LIN {X 0,Y 400.14,Z 423.786,A -85,B 0,C 180,E1 -11270.146,E2 -11270.146} C_VEL
LIN {X 0,Y 399.174,Z 418.317,A -85,B 0,C 180,E1 -11270.323,E2 -11270.323} C_VEL
LIN {X 0,Y 400.535,Z 402.133,A -85,B 0,C 180,E1 -11273.803,E2 -11273.803} C_VEL
LIN {X 0,Y 400.601,Z 399.085,A -85,B 0,C 180,E1 -11274.478,E2 -11274.478} C_VEL
LIN {X 0,Y 398.361,Z 387.399,A -85,B 0,C 180,E1 -11277.304,E2 -11277.304} C_VEL
LIN {X 0,Y 397.149,Z 382.018,A -85,B 0,C 180,E1 -11278.687,E2 -11278.687} C_VEL
LIN {X 0,Y 397.084,Z 382.025,A -85,B 0,C 180,E1 -11282.072,E2 -11282.072} C_VEL
LIN {X 0,Y 397.125,Z 382.02,A -85,B 0,C 180,E1 -11285.504,E2 -11285.504} C_VEL
LIN {X 0,Y 397.136,Z 382.02,A -85,B 0,C 180,E1 -11288.862,E2 -11288.862} C_VEL
LIN {X 0,Y 397.074,Z 382.025,A -85,B 0,C 180,E1 -11292.268,E2 -11292.268} C_VEL
LIN {X 0,Y 397.092,Z 382.023,A -85,B 0,C 180,E1 -11295.069,E2 -11295.069} C_VEL
LIN {X 0,Y 397.071,Z 382.022,A -85,B 0,C 180,E1 -11298.022,E2 -11298.022} C_VEL
LIN {X 0,Y 397.134,Z 382.018,A -85,B 0,C 180,E1 -11301.139,E2 -11301.139} C_VEL
LIN {X 0,Y 397.125,Z 382.018,A -85,B 0,C 180,E1 -11304.497,E2 -11304.497} C_VEL
LIN {X 0,Y 397.084,Z 382.02,A -85,B 0,C 180,E1 -11307.929,E2 -11307.929} C_VEL
LIN {X 0,Y 397.128,Z 382.015,A -85,B 0,C 180,E1 -11311.457,E2 -11311.457} C_VEL
LIN {X 0,Y 397.158,Z 382.011,A -85,B 0,C 180,E1 -11314.488,E2 -11314.488} C_VEL
LIN {X 0,Y 397.115,Z 382.014,A -85,B 0,C 180,E1 -11318.183,E2 -11318.183} C_VEL
LIN {X 0,Y 397.168,Z 382.003,A -85,B 0,C 180,E1 -11321.427,E2 -11321.427} C_VEL
LIN {X 0,Y 397.185,Z 382.005,A -85,B 0,C 180,E1 -11324.608,E2 -11324.608} C_VEL
LIN {X 0,Y 397.225,Z 382.004,A -85,B 0,C 180,E1 -11327.742,E2 -11327.742} C_VEL
LIN {X 0,Y 397.401,Z 381.985,A -85,B 0,C 180,E1 -11332.041,E2 -11332.041} C_VEL
LIN {X 0,Y 397.26,Z 381.999,A -85,B 0,C 180,E1 -11334.925,E2 -11334.925} C_VEL
LIN {X 0,Y 397.455,Z 381.973,A -85,B 0,C 180,E1 -11337.973,E2 -11337.973} C_VEL
LIN {X 0,Y 397.585,Z 381.959,A -85,B 0,C 180,E1 -11340,E2 -11340} C_VEL
LIN {X 0,Y 397.382,Z 381.983,A -85,B 0,C 180,E1 -11343.041,E2 -11343.041} C_VEL
LIN {X 0,Y 397.37,Z 381.983,A -85,B 0,C 180,E1 -11347.112,E2 -11347.112} C_VEL
LIN {X 0,Y 397.224,Z 382.008,A -85,B 0,C 180,E1 -11350.191,E2 -11350.191} C_VEL
LIN {X 0,Y 397.233,Z 382.005,A -85,B 0,C 180,E1 -11353.321,E2 -11353.321} C_VEL
LIN {X 0,Y 397.188,Z 382.01,A -85,B 0,C 180,E1 -11357.155,E2 -11357.155} C_VEL
LIN {X 0,Y 397.109,Z 382.019,A -85,B 0,C 180,E1 -11360.73,E2 -11360.73} C_VEL
LIN {X 0,Y 397.139,Z 382.015,A -85,B 0,C 180,E1 -11364.018,E2 -11364.018} C_VEL
LIN {X 0,Y 397.231,Z 382.12,A -85,B 0,C 180,E1 -11367.209,E2 -11367.209} C_VEL
LIN {X 0,Y 399.17,Z 392.144,A -85,B 0,C 180,E1 -11370.004,E2 -11370.004} C_VEL
LIN {X 0,Y 399.737,Z 396.779,A -85,B 0,C 180,E1 -11371.242,E2 -11371.242} C_VEL
LIN {X 0,Y 399.607,Z 398.872,A -85,B 0,C 180,E1 -11371.771,E2 -11371.771} C_VEL
LIN {X 0,Y 404.077,Z 419.363,A -85,B 0,C 180,E1 -11372.445,E2 -11372.445} C_VEL
LIN {X 0,Y 404.272,Z 424.24,A -85,B 0,C 180,E1 -11372.552,E2 -11372.552} C_VEL
LIN {X 0,Y 402.86,Z 505.983,A -85,B 0,C 180,E1 -11374.111,E2 -11374.111} C_VEL
LIN {X 0,Y 402.397,Z 518.755,A -85,B 0,C 180,E1 -11374.545,E2 -11374.545} C_VEL
LIN {X 0,Y 401.764,Z 531.63,A -85,B 0,C 180,E1 -11375.191,E2 -11375.191} C_VEL
LIN {X 0,Y 400.956,Z 543.977,A -85,B 0,C 180,E1 -11376.043,E2 -11376.043} C_VEL
LIN {X 0,Y 400.163,Z 554.558,A -85,B 0,C 180,E1 -11376.98,E2 -11376.98} C_VEL
LIN {X 0,Y 399.29,Z 565.476,A -85,B 0,C 180,E1 -11378.188,E2 -11378.188} C_VEL
LIN {X 0,Y 398.415,Z 574.461,A -85,B 0,C 180,E1 -11379.423,E2 -11379.423} C_VEL
LIN {X 0,Y 397.649,Z 582.829,A -85,B 0,C 180,E1 -11380.839,E2 -11380.839} C_VEL
LIN {X 0,Y 397.067,Z 589.697,A -85,B 0,C 180,E1 -11382.268,E2 -11382.268} C_VEL
LIN {X 0,Y 396.606,Z 595.356,A -85,B 0,C 180,E1 -11383.717,E2 -11383.717} C_VEL
LIN {X 0,Y 396.229,Z 599.96,A -85,B 0,C 180,E1 -11385.194,E2 -11385.194} C_VEL
LIN {X 0,Y 395.96,Z 603.578,A -85,B 0,C 180,E1 -11386.696,E2 -11386.696} C_VEL
LIN {X 0,Y 395.753,Z 606.265,A -85,B 0,C 180,E1 -11388.233,E2 -11388.233} C_VEL
LIN {X 0,Y 395.599,Z 608.354,A -85,B 0,C 180,E1 -11390.24,E2 -11390.24} C_VEL
LIN {X 0,Y 395.556,Z 608.831,A -85,B 0,C 180,E1 -11391.547,E2 -11391.547} C_VEL
LIN {X 0,Y 395.557,Z 608.577,A -85,B 0,C 180,E1 -11393.086,E2 -11393.086} C_VEL
LIN {X 0,Y 395.648,Z 607.213,A -85,B 0,C 180,E1 -11394.797,E2 -11394.797} C_VEL
LIN {X 0,Y 395.849,Z 604.514,A -85,B 0,C 180,E1 -11396.606,E2 -11396.606} C_VEL
LIN {X 0,Y 396.124,Z 600.493,A -85,B 0,C 180,E1 -11398.388,E2 -11398.388} C_VEL
LIN {X 0,Y 396.495,Z 594.51,A -85,B 0,C 180,E1 -11400.29,E2 -11400.29} C_VEL
LIN {X 0,Y 397.001,Z 588.053,A -85,B 0,C 180,E1 -11401.873,E2 -11401.873} C_VEL
LIN {X 0,Y 397.556,Z 581.327,A -85,B 0,C 180,E1 -11403.204,E2 -11403.204} C_VEL
LIN {X 0,Y 398.312,Z 571.9,A -85,B 0,C 180,E1 -11404.714,E2 -11404.714} C_VEL
LIN {X 0,Y 399.125,Z 562.154,A -85,B 0,C 180,E1 -11405.97,E2 -11405.97} C_VEL
LIN {X 0,Y 399.932,Z 551.066,A -85,B 0,C 180,E1 -11407.119,E2 -11407.119} C_VEL
LIN {X 0,Y 400.708,Z 539.338,A -85,B 0,C 180,E1 -11408.069,E2 -11408.069} C_VEL
LIN {X 0,Y 401.313,Z 527.263,A -85,B 0,C 180,E1 -11408.825,E2 -11408.825} C_VEL
LIN {X 0,Y 401.878,Z 514.644,A -85,B 0,C 180,E1 -11409.393,E2 -11409.393} C_VEL
LIN {X 0,Y 402.234,Z 500.536,A -85,B 0,C 180,E1 -11409.794,E2 -11409.794} C_VEL
LIN {X 0,Y 403.386,Z 420.013,A -85,B 0,C 180,E1 -11411.293,E2 -11411.293} C_VEL
LIN {X 0,Y 399.172,Z 398.042,A -85,B 0,C 180,E1 -11411.944,E2 -11411.944} C_VEL
LIN {X 0,Y 399.24,Z 393.33,A -85,B 0,C 180,E1 -11413.114,E2 -11413.114} C_VEL
LIN {X 0,Y 397.325,Z 382.653,A -85,B 0,C 180,E1 -11415.923,E2 -11415.923} C_VEL
LIN {X 0,Y 397.222,Z 382.008,A -85,B 0,C 180,E1 -11416.152,E2 -11416.152} C_VEL
LIN {X 0,Y 396.586,Z 382.088,A -85,B 0,C 180,E1 -11416.997,E2 -11416.997} C_VEL
LIN {X 0,Y 393.705,Z 382.445,A -85,B 0,C 180,E1 -11418.371,E2 -11418.371} C_VEL
LIN {X 0,Y 391.27,Z 382.745,A -85,B 0,C 180,E1 -11419.482,E2 -11419.482} C_VEL
LIN {X 0,Y 390.265,Z 382.873,A -85,B 0,C 180,E1 -11420.341,E2 -11420.341} C_VEL
LIN {X 0,Y 390.206,Z 382.88,A -85,B 0,C 180,E1 -11420.632,E2 -11420.632} C_VEL
LIN {X 0,Y 390.304,Z 382.864,A -85,B 0,C 180,E1 -11423.796,E2 -11423.796} C_VEL
LIN {X 0,Y 390.423,Z 382.851,A -85,B 0,C 180,E1 -11427.935,E2 -11427.935} C_VEL
LIN {X 0,Y 390.552,Z 382.835,A -85,B 0,C 180,E1 -11429.999,E2 -11429.999} C_VEL
LIN {X 0,Y 390.318,Z 382.862,A -85,B 0,C 180,E1 -11433.095,E2 -11433.095} C_VEL
LIN {X 0,Y 390.333,Z 382.866,A -85,B 0,C 180,E1 -11436.2,E2 -11436.2} C_VEL
LIN {X 0,Y 390.317,Z 382.867,A -85,B 0,C 180,E1 -11438.281,E2 -11438.281} C_VEL
LIN {X 0,Y 390.172,Z 382.882,A -85,B 0,C 180,E1 -11442.482,E2 -11442.482} C_VEL
LIN {X 0,Y 390.145,Z 382.886,A -85,B 0,C 180,E1 -11445.675,E2 -11445.675} C_VEL
LIN {X 0,Y 390.106,Z 382.888,A -85,B 0,C 180,E1 -11448.92,E2 -11448.92} C_VEL
LIN {X 0,Y 390.036,Z 382.9,A -85,B 0,C 180,E1 -11452.233,E2 -11452.233} C_VEL
LIN {X 0,Y 390.117,Z 382.892,A -85,B 0,C 180,E1 -11455.742,E2 -11455.742} C_VEL
LIN {X 0,Y 390.07,Z 382.893,A -85,B 0,C 180,E1 -11459.107,E2 -11459.107} C_VEL
LIN {X 0,Y 390.052,Z 382.895,A -85,B 0,C 180,E1 -11462.719,E2 -11462.719} C_VEL
LIN {X 0,Y 390.053,Z 382.899,A -85,B 0,C 180,E1 -11465.824,E2 -11465.824} C_VEL
LIN {X 0,Y 390.07,Z 382.895,A -85,B 0,C 180,E1 -11469.218,E2 -11469.218} C_VEL
LIN {X 0,Y 390.076,Z 382.892,A -85,B 0,C 180,E1 -11472.379,E2 -11472.379} C_VEL
LIN {X 0,Y 390.134,Z 383.038,A -85,B 0,C 180,E1 -11475.045,E2 -11475.045} C_VEL
LIN {X 0,Y 391.764,Z 391.926,A -85,B 0,C 180,E1 -11477.023,E2 -11477.023} C_VEL
LIN {X 0,Y 391.869,Z 396.801,A -85,B 0,C 180,E1 -11478.061,E2 -11478.061} C_VEL
LIN {X 0,Y 396.111,Z 421.486,A -85,B 0,C 180,E1 -11478.798,E2 -11478.798} C_VEL
LIN {X 0,Y 394.513,Z 506.118,A -85,B 0,C 180,E1 -11480.565,E2 -11480.565} C_VEL
LIN {X 0,Y 394.042,Z 519.35,A -85,B 0,C 180,E1 -11481.045,E2 -11481.045} C_VEL
LIN {X 0,Y 393.451,Z 532.156,A -85,B 0,C 180,E1 -11481.727,E2 -11481.727} C_VEL
LIN {X 0,Y 392.826,Z 543.595,A -85,B 0,C 180,E1 -11482.534,E2 -11482.534} C_VEL
LIN {X 0,Y 392.073,Z 555.083,A -85,B 0,C 180,E1 -11483.574,E2 -11483.574} C_VEL
LIN {X 0,Y 391.358,Z 565.608,A -85,B 0,C 180,E1 -11484.767,E2 -11484.767} C_VEL
LIN {X 0,Y 390.619,Z 575.13,A -85,B 0,C 180,E1 -11486.099,E2 -11486.099} C_VEL
LIN {X 0,Y 390.034,Z 583.947,A -85,B 0,C 180,E1 -11487.635,E2 -11487.635} C_VEL
LIN {X 0,Y 389.517,Z 590.564,A -85,B 0,C 180,E1 -11489.054,E2 -11489.054} C_VEL
LIN {X 0,Y 389.113,Z 597.059,A -85,B 0,C 180,E1 -11490.813,E2 -11490.813} C_VEL
LIN {X 0,Y 388.883,Z 601.347,A -85,B 0,C 180,E1 -11492.314,E2 -11492.314} C_VEL
LIN {X 0,Y 388.659,Z 605.419,A -85,B 0,C 180,E1 -11494.279,E2 -11494.279} C_VEL
LIN {X 0,Y 388.558,Z 607.024,A -85,B 0,C 180,E1 -11495.417,E2 -11495.417} C_VEL
LIN {X 0,Y 388.467,Z 608.568,A -85,B 0,C 180,E1 -11497.315,E2 -11497.315} C_VEL
LIN {X 0,Y 388.461,Z 608.799,A -85,B 0,C 180,E1 -11498.787,E2 -11498.787} C_VEL
LIN {X 0,Y 388.561,Z 608.285,A -85,B 0,C 180,E1 -11500.137,E2 -11500.137} C_VEL
LIN {X 0,Y 388.72,Z 606.239,A -85,B 0,C 180,E1 -11502.1,E2 -11502.1} C_VEL
LIN {X 0,Y 388.952,Z 603.258,A -85,B 0,C 180,E1 -11503.785,E2 -11503.785} C_VEL
LIN {X 0,Y 389.24,Z 599.364,A -85,B 0,C 180,E1 -11505.358,E2 -11505.358} C_VEL
LIN {X 0,Y 389.821,Z 593.33,A -85,B 0,C 180,E1 -11507.175,E2 -11507.175} C_VEL
LIN {X 0,Y 390.466,Z 586.19,A -85,B 0,C 180,E1 -11508.843,E2 -11508.843} C_VEL
LIN {X 0,Y 391.265,Z 577.579,A -85,B 0,C 180,E1 -11510.436,E2 -11510.436} C_VEL
LIN {X 0,Y 392.122,Z 568.734,A -85,B 0,C 180,E1 -11511.756,E2 -11511.756} C_VEL
LIN {X 0,Y 392.956,Z 559.087,A -85,B 0,C 180,E1 -11512.937,E2 -11512.937} C_VEL
LIN {X 0,Y 393.913,Z 548.424,A -85,B 0,C 180,E1 -11513.983,E2 -11513.983} C_VEL
LIN {X 0,Y 394.785,Z 536.723,A -85,B 0,C 180,E1 -11514.893,E2 -11514.893} C_VEL
LIN {X 0,Y 395.478,Z 524.195,A -85,B 0,C 180,E1 -11515.641,E2 -11515.641} C_VEL
LIN {X 0,Y 396.088,Z 511.196,A -85,B 0,C 180,E1 -11516.185,E2 -11516.185} C_VEL
LIN {X 0,Y 396.467,Z 497.95,A -85,B 0,C 180,E1 -11516.538,E2 -11516.538} C_VEL
LIN {X 0,Y 398.352,Z 421.721,A -85,B 0,C 180,E1 -11518.2,E2 -11518.2} C_VEL
LIN {X 0,Y 395.108,Z 405.743,A -85,B 0,C 180,E1 -11518.816,E2 -11518.816} C_VEL
LIN {X 0,Y 393.13,Z 397.845,A -85,B 0,C 180,E1 -11519.162,E2 -11519.162} C_VEL
LIN {X 0,Y 392.414,Z 391.776,A -85,B 0,C 180,E1 -11520.513,E2 -11520.513} C_VEL
LIN {X 0,Y 390.363,Z 382.864,A -85,B 0,C 180,E1 -11522.58,E2 -11522.58} C_VEL
LIN {X 0,Y 390.319,Z 382.869,A -85,B 0,C 180,E1 -11526.202,E2 -11526.202} C_VEL
LIN {X 0,Y 390.304,Z 382.867,A -85,B 0,C 180,E1 -11528.282,E2 -11528.282} C_VEL
LIN {X 0,Y 390.167,Z 382.884,A -85,B 0,C 180,E1 -11532.483,E2 -11532.483} C_VEL
LIN {X 0,Y 390.133,Z 382.89,A -85,B 0,C 180,E1 -11535.677,E2 -11535.677} C_VEL
LIN {X 0,Y 390.109,Z 382.891,A -85,B 0,C 180,E1 -11538.922,E2 -11538.922} C_VEL
LIN {X 0,Y 390.104,Z 382.892,A -85,B 0,C 180,E1 -11542.23,E2 -11542.23} C_VEL
LIN {X 0,Y 390.11,Z 382.893,A -85,B 0,C 180,E1 -11545.744,E2 -11545.744} C_VEL
LIN {X 0,Y 390.056,Z 382.898,A -85,B 0,C 180,E1 -11549.11,E2 -11549.11} C_VEL
LIN {X 0,Y 390.046,Z 382.898,A -85,B 0,C 180,E1 -11552.721,E2 -11552.721} C_VEL
LIN {X 0,Y 390.048,Z 382.9,A -85,B 0,C 180,E1 -11555.827,E2 -11555.827} C_VEL
LIN {X 0,Y 390.064,Z 382.897,A -85,B 0,C 180,E1 -11559.22,E2 -11559.22} C_VEL
LIN {X 0,Y 390.037,Z 382.898,A -85,B 0,C 180,E1 -11562.376,E2 -11562.376} C_VEL
LIN {X 0,Y 390.041,Z 382.901,A -85,B 0,C 180,E1 -11565.356,E2 -11565.356} C_VEL
LIN {X 0,Y 390.026,Z 382.9,A -85,B 0,C 180,E1 -11568.188,E2 -11568.188} C_VEL
LIN {X 0,Y 390.086,Z 382.895,A -85,B 0,C 180,E1 -11570.909,E2 -11570.909} C_VEL
LIN {X 0,Y 390.081,Z 382.897,A -85,B 0,C 180,E1 -11574.795,E2 -11574.795} C_VEL
LIN {X 0,Y 390.045,Z 382.901,A -85,B 0,C 180,E1 -11578.5,E2 -11578.5} C_VEL
LIN {X 0,Y 390.16,Z 382.993,A -85,B 0,C 180,E1 -11581.612,E2 -11581.612} C_VEL
LIN {X 0,Y 392.272,Z 393.449,A -85,B 0,C 180,E1 -11584.136,E2 -11584.136} C_VEL
LIN {X 0,Y 393.422,Z 400.338,A -85,B 0,C 180,E1 -11585.742,E2 -11585.742} C_VEL
LIN {X 0,Y 392.335,Z 413.865,A -85,B 0,C 180,E1 -11588.669,E2 -11588.669} C_VEL
LIN {X 0,Y 392.214,Z 415.631,A -85,B 0,C 180,E1 -11589.049,E2 -11589.049} C_VEL
LIN {X 0,Y 395.398,Z 433.743,A -85,B 0,C 180,E1 -11589.737,E2 -11589.737} C_VEL
LIN {X 0,Y 397.27,Z 448.692,A -85,B 0,C 180,E1 -11590.226,E2 -11590.226} C_VEL
LIN {X 0,Y 395.443,Z 528.264,A -85,B 0,C 180,E1 -11592.015,E2 -11592.015} C_VEL
LIN {X 0,Y 394.717,Z 541.627,A -85,B 0,C 180,E1 -11592.516,E2 -11592.516} C_VEL
LIN {X 0,Y 394.011,Z 553.409,A -85,B 0,C 180,E1 -11593.152,E2 -11593.152} C_VEL
LIN {X 0,Y 392.984,Z 567.466,A -85,B 0,C 180,E1 -11594.175,E2 -11594.175} C_VEL
LIN {X 0,Y 392.109,Z 578.543,A -85,B 0,C 180,E1 -11595.204,E2 -11595.204} C_VEL
LIN {X 0,Y 391.257,Z 589.501,A -85,B 0,C 180,E1 -11596.497,E2 -11596.497} C_VEL
LIN {X 0,Y 390.544,Z 598.401,A -85,B 0,C 180,E1 -11597.794,E2 -11597.794} C_VEL
LIN {X 0,Y 389.885,Z 605.74,A -85,B 0,C 180,E1 -11599.091,E2 -11599.091} C_VEL
LIN {X 0,Y 389.38,Z 612.957,A -85,B 0,C 180,E1 -11600.653,E2 -11600.653} C_VEL
LIN {X 0,Y 389.024,Z 618.699,A -85,B 0,C 180,E1 -11602.214,E2 -11602.214} C_VEL
LIN {X 0,Y 388.791,Z 623.351,A -85,B 0,C 180,E1 -11603.833,E2 -11603.833} C_VEL
LIN {X 0,Y 388.742,Z 625.589,A -85,B 0,C 180,E1 -11604.815,E2 -11604.815} C_VEL
LIN {X 0,Y 388.7,Z 627.529,A -85,B 0,C 180,E1 -11605.854,E2 -11605.854} C_VEL
LIN {X 0,Y 388.636,Z 629.032,A -85,B 0,C 180,E1 -11606.891,E2 -11606.891} C_VEL
LIN {X 0,Y 388.662,Z 630.082,A -85,B 0,C 180,E1 -11607.929,E2 -11607.929} C_VEL
LIN {X 0,Y 388.703,Z 630.735,A -85,B 0,C 180,E1 -11608.965,E2 -11608.965} C_VEL
LIN {X 0,Y 388.707,Z 630.995,A -85,B 0,C 180,E1 -11610.001,E2 -11610.001} C_VEL
LIN {X 0,Y 388.703,Z 630.844,A -85,B 0,C 180,E1 -11611.037,E2 -11611.037} C_VEL
LIN {X 0,Y 388.661,Z 630.258,A -85,B 0,C 180,E1 -11612.074,E2 -11612.074} C_VEL
LIN {X 0,Y 388.7,Z 627.898,A -85,B 0,C 180,E1 -11614.149,E2 -11614.149} C_VEL
LIN {X 0,Y 388.729,Z 624.881,A -85,B 0,C 180,E1 -11615.757,E2 -11615.757} C_VEL
LIN {X 0,Y 388.939,Z 621.035,A -85,B 0,C 180,E1 -11617.268,E2 -11617.268} C_VEL
LIN {X 0,Y 389.264,Z 615.949,A -85,B 0,C 180,E1 -11618.829,E2 -11618.829} C_VEL
LIN {X 0,Y 389.778,Z 609.569,A -85,B 0,C 180,E1 -11620.389,E2 -11620.389} C_VEL
LIN {X 0,Y 390.471,Z 601.583,A -85,B 0,C 180,E1 -11621.947,E2 -11621.947} C_VEL
LIN {X 0,Y 391.29,Z 593.46,A -85,B 0,C 180,E1 -11623.24,E2 -11623.24} C_VEL
LIN {X 0,Y 392.062,Z 583.568,A -85,B 0,C 180,E1 -11624.536,E2 -11624.536} C_VEL
LIN {X 0,Y 393.047,Z 572.516,A -85,B 0,C 180,E1 -11625.692,E2 -11625.692} C_VEL
LIN {X 0,Y 393.949,Z 561.71,A -85,B 0,C 180,E1 -11626.586,E2 -11626.586} C_VEL
LIN {X 0,Y 394.872,Z 548.732,A -85,B 0,C 180,E1 -11627.413,E2 -11627.413} C_VEL
LIN {X 0,Y 395.55,Z 536.29,A -85,B 0,C 180,E1 -11627.983,E2 -11627.983} C_VEL
LIN {X 0,Y 396.139,Z 523.542,A -85,B 0,C 180,E1 -11628.356,E2 -11628.356} C_VEL
LIN {X 0,Y 397.249,Z 447.452,A -85,B 0,C 180,E1 -11629.829,E2 -11629.829} C_VEL
LIN {X 0,Y 393.184,Z 422.506,A -85,B 0,C 180,E1 -11630.579,E2 -11630.579} C_VEL
LIN {X 0,Y 392.324,Z 418.111,A -85,B 0,C 180,E1 -11630.732,E2 -11630.732} C_VEL
LIN {X 0,Y 393.764,Z 402.116,A -85,B 0,C 180,E1 -11634.238,E2 -11634.238} C_VEL
LIN {X 0,Y 392.703,Z 395.034,A -85,B 0,C 180,E1 -11635.944,E2 -11635.944} C_VEL
LIN {X 0,Y 390.521,Z 384.688,A -85,B 0,C 180,E1 -11638.565,E2 -11638.565} C_VEL
LIN {X 0,Y 390.11,Z 382.896,A -85,B 0,C 180,E1 -11639.043,E2 -11639.043} C_VEL
LIN {X 0,Y 390.048,Z 382.902,A -85,B 0,C 180,E1 -11642.722,E2 -11642.722} C_VEL
LIN {X 0,Y 390.061,Z 382.899,A -85,B 0,C 180,E1 -11645.826,E2 -11645.826} C_VEL
LIN {X 0,Y 390.076,Z 382.902,A -85,B 0,C 180,E1 -11649.219,E2 -11649.219} C_VEL
LIN {X 0,Y 390.048,Z 382.901,A -85,B 0,C 180,E1 -11652.375,E2 -11652.375} C_VEL
LIN {X 0,Y 390.05,Z 382.901,A -85,B 0,C 180,E1 -11655.355,E2 -11655.355} C_VEL
LIN {X 0,Y 390.036,Z 382.899,A -85,B 0,C 180,E1 -11658.187,E2 -11658.187} C_VEL
LIN {X 0,Y 390.094,Z 382.894,A -85,B 0,C 180,E1 -11660.908,E2 -11660.908} C_VEL
LIN {X 0,Y 390.091,Z 382.895,A -85,B 0,C 180,E1 -11664.794,E2 -11664.794} C_VEL
LIN {X 0,Y 390.03,Z 382.902,A -85,B 0,C 180,E1 -11668.496,E2 -11668.496} C_VEL
LIN {X 0,Y 390.123,Z 382.888,A -85,B 0,C 180,E1 -11672.07,E2 -11672.07} C_VEL
LIN {X 0,Y 390.085,Z 382.892,A -85,B 0,C 180,E1 -11675.52,E2 -11675.52} C_VEL
LIN {X 0,Y 390.069,Z 382.897,A -85,B 0,C 180,E1 -11678.879,E2 -11678.879} C_VEL
LIN {X 0,Y 390.134,Z 382.882,A -85,B 0,C 180,E1 -11682.167,E2 -11682.167} C_VEL
LIN {X 0,Y 390.15,Z 382.877,A -85,B 0,C 180,E1 -11685.393,E2 -11685.393} C_VEL
LIN {X 0,Y 390.154,Z 382.881,A -85,B 0,C 180,E1 -11688.571,E2 -11688.571} C_VEL
LIN {X 0,Y 390.35,Z 382.863,A -85,B 0,C 180,E1 -11691.994,E2 -11691.994} C_VEL
LIN {X 0,Y 390.233,Z 382.875,A -85,B 0,C 180,E1 -11694.834,E2 -11694.834} C_VEL
LIN {X 0,Y 390.424,Z 382.848,A -85,B 0,C 180,E1 -11697.937,E2 -11697.937} C_VEL
LIN {X 0,Y 390.554,Z 382.834,A -85,B 0,C 180,E1 -11700,E2 -11700} C_VEL
LIN {X 0,Y 390.316,Z 382.863,A -85,B 0,C 180,E1 -11703.097,E2 -11703.097} C_VEL
LIN {X 0,Y 390.316,Z 382.861,A -85,B 0,C 180,E1 -11706.636,E2 -11706.636} C_VEL
LIN {X 0,Y 390.211,Z 382.878,A -85,B 0,C 180,E1 -11709.329,E2 -11709.329} C_VEL
LIN {X 0,Y 390.201,Z 382.882,A -85,B 0,C 180,E1 -11713.438,E2 -11713.438} C_VEL
LIN {X 0,Y 390.155,Z 382.888,A -85,B 0,C 180,E1 -11717.308,E2 -11717.308} C_VEL
LIN {X 0,Y 390.094,Z 382.893,A -85,B 0,C 180,E1 -11720.47,E2 -11720.47} C_VEL
LIN {X 0,Y 390.096,Z 382.892,A -85,B 0,C 180,E1 -11723.351,E2 -11723.351} C_VEL
LIN {X 0,Y 390.14,Z 382.932,A -85,B 0,C 180,E1 -11726.839,E2 -11726.839} C_VEL
LIN {X 0,Y 392.089,Z 392.334,A -85,B 0,C 180,E1 -11729.533,E2 -11729.533} C_VEL
LIN {X 0,Y 392.827,Z 397.002,A -85,B 0,C 180,E1 -11730.821,E2 -11730.821} C_VEL
LIN {X 0,Y 392.788,Z 399.153,A -85,B 0,C 180,E1 -11731.37,E2 -11731.37} C_VEL
LIN {X 0,Y 397.255,Z 419.381,A -85,B 0,C 180,E1 -11732.056,E2 -11732.056} C_VEL
LIN {X 0,Y 397.726,Z 422.904,A -85,B 0,C 180,E1 -11732.156,E2 -11732.156} C_VEL
LIN {X 0,Y 396.164,Z 506.525,A -85,B 0,C 180,E1 -11733.784,E2 -11733.784} C_VEL
LIN {X 0,Y 395.612,Z 520.228,A -85,B 0,C 180,E1 -11734.268,E2 -11734.268} C_VEL
LIN {X 0,Y 394.981,Z 532.849,A -85,B 0,C 180,E1 -11734.934,E2 -11734.934} C_VEL
LIN {X 0,Y 394.137,Z 544.815,A -85,B 0,C 180,E1 -11735.788,E2 -11735.788} C_VEL
LIN {X 0,Y 393.267,Z 555.993,A -85,B 0,C 180,E1 -11736.813,E2 -11736.813} C_VEL
LIN {X 0,Y 392.375,Z 566.25,A -85,B 0,C 180,E1 -11737.99,E2 -11737.99} C_VEL
LIN {X 0,Y 391.328,Z 576.363,A -85,B 0,C 180,E1 -11739.442,E2 -11739.442} C_VEL
LIN {X 0,Y 390.555,Z 584.556,A -85,B 0,C 180,E1 -11740.904,E2 -11740.904} C_VEL
LIN {X 0,Y 389.967,Z 591.163,A -85,B 0,C 180,E1 -11742.36,E2 -11742.36} C_VEL
LIN {X 0,Y 389.509,Z 596.46,A -85,B 0,C 180,E1 -11743.801,E2 -11743.801} C_VEL
LIN {X 0,Y 389.139,Z 600.644,A -85,B 0,C 180,E1 -11745.221,E2 -11745.221} C_VEL
LIN {X 0,Y 388.885,Z 603.883,A -85,B 0,C 180,E1 -11746.626,E2 -11746.626} C_VEL
LIN {X 0,Y 388.692,Z 606.283,A -85,B 0,C 180,E1 -11748.009,E2 -11748.009} C_VEL
LIN {X 0,Y 388.57,Z 607.982,A -85,B 0,C 180,E1 -11749.434,E2 -11749.434} C_VEL
LIN {X 0,Y 388.461,Z 608.966,A -85,B 0,C 180,E1 -11751.074,E2 -11751.074} C_VEL
LIN {X 0,Y 388.462,Z 608.931,A -85,B 0,C 180,E1 -11752.754,E2 -11752.754} C_VEL
LIN {X 0,Y 388.533,Z 607.627,A -85,B 0,C 180,E1 -11754.63,E2 -11754.63} C_VEL
LIN {X 0,Y 388.678,Z 605.384,A -85,B 0,C 180,E1 -11756.281,E2 -11756.281} C_VEL
LIN {X 0,Y 389.015,Z 601.591,A -85,B 0,C 180,E1 -11758.115,E2 -11758.115} C_VEL
LIN {X 0,Y 389.269,Z 597.335,A -85,B 0,C 180,E1 -11759.633,E2 -11759.633} C_VEL
LIN {X 0,Y 389.822,Z 590.691,A -85,B 0,C 180,E1 -11761.46,E2 -11761.46} C_VEL
LIN {X 0,Y 390.383,Z 583.721,A -85,B 0,C 180,E1 -11762.961,E2 -11762.961} C_VEL
LIN {X 0,Y 391.071,Z 575.19,A -85,B 0,C 180,E1 -11764.448,E2 -11764.448} C_VEL
LIN {X 0,Y 391.856,Z 565.888,A -85,B 0,C 180,E1 -11765.764,E2 -11765.764} C_VEL
LIN {X 0,Y 392.753,Z 555.395,A -85,B 0,C 180,E1 -11766.955,E2 -11766.955} C_VEL
LIN {X 0,Y 393.508,Z 544.205,A -85,B 0,C 180,E1 -11767.971,E2 -11767.971} C_VEL
LIN {X 0,Y 394.249,Z 531.903,A -85,B 0,C 180,E1 -11768.841,E2 -11768.841} C_VEL
LIN {X 0,Y 394.888,Z 518.564,A -85,B 0,C 180,E1 -11769.522,E2 -11769.522} C_VEL
LIN {X 0,Y 395.367,Z 505.398,A -85,B 0,C 180,E1 -11769.972,E2 -11769.972} C_VEL
LIN {X 0,Y 396.682,Z 421.155,A -85,B 0,C 180,E1 -11771.587,E2 -11771.587} C_VEL
LIN {X 0,Y 392.264,Z 398.293,A -85,B 0,C 180,E1 -11772.266,E2 -11772.266} C_VEL
LIN {X 0,Y 392.205,Z 394.066,A -85,B 0,C 180,E1 -11773.338,E2 -11773.338} C_VEL
LIN {X 0,Y 390.181,Z 382.885,A -85,B 0,C 180,E1 -11776.357,E2 -11776.357} C_VEL
LIN {X 0,Y 390.174,Z 382.881,A -85,B 0,C 180,E1 -11779.622,E2 -11779.622} C_VEL
LIN {X 0,Y 390.206,Z 382.88,A -85,B 0,C 180,E1 -11780.632,E2 -11780.632} C_VEL
LIN {X 0,Y 389.609,Z 382.961,A -85,B 0,C 180,E1 -11781.495,E2 -11781.495} C_VEL
LIN {X 0,Y 386.797,Z 383.312,A -85,B 0,C 180,E1 -11782.897,E2 -11782.897} C_VEL
LIN {X 0,Y 384.343,Z 383.612,A -85,B 0,C 180,E1 -11784.03,E2 -11784.03} C_VEL
LIN {X 0,Y 383.239,Z 383.746,A -85,B 0,C 180,E1 -11784.906,E2 -11784.906} C_VEL
LIN {X 0,Y 383.125,Z 383.758,A -85,B 0,C 180,E1 -11785.204,E2 -11785.204} C_VEL
LIN {X 0,Y 383.39,Z 383.726,A -85,B 0,C 180,E1 -11787.898,E2 -11787.898} C_VEL
LIN {X 0,Y 383.522,Z 383.711,A -85,B 0,C 180,E1 -11789.999,E2 -11789.999} C_VEL
LIN {X 0,Y 383.254,Z 383.742,A -85,B 0,C 180,E1 -11793.152,E2 -11793.152} C_VEL
LIN {X 0,Y 383.29,Z 383.743,A -85,B 0,C 180,E1 -11796.315,E2 -11796.315} C_VEL
LIN {X 0,Y 383.262,Z 383.744,A -85,B 0,C 180,E1 -11798.434,E2 -11798.434} C_VEL
LIN {X 0,Y 383.099,Z 383.763,A -85,B 0,C 180,E1 -11801.641,E2 -11801.641} C_VEL
LIN {X 0,Y 383.114,Z 383.759,A -85,B 0,C 180,E1 -11804.88,E2 -11804.88} C_VEL
LIN {X 0,Y 383.09,Z 383.767,A -85,B 0,C 180,E1 -11808.171,E2 -11808.171} C_VEL
LIN {X 0,Y 382.991,Z 383.777,A -85,B 0,C 180,E1 -11811.529,E2 -11811.529} C_VEL
LIN {X 0,Y 383.049,Z 383.767,A -85,B 0,C 180,E1 -11814.959,E2 -11814.959} C_VEL
LIN {X 0,Y 383.049,Z 383.768,A -85,B 0,C 180,E1 -11818.49,E2 -11818.49} C_VEL
LIN {X 0,Y 383.034,Z 383.771,A -85,B 0,C 180,E1 -11822.145,E2 -11822.145} C_VEL
LIN {X 0,Y 383.023,Z 383.774,A -85,B 0,C 180,E1 -11825.954,E2 -11825.954} C_VEL
LIN {X 0,Y 383.017,Z 383.778,A -85,B 0,C 180,E1 -11829.586,E2 -11829.586} C_VEL
LIN {X 0,Y 383.026,Z 383.77,A -85,B 0,C 180,E1 -11832.781,E2 -11832.781} C_VEL
LIN {X 0,Y 383.057,Z 383.853,A -85,B 0,C 180,E1 -11834.853,E2 -11834.853} C_VEL
LIN {X 0,Y 384.779,Z 393.094,A -85,B 0,C 180,E1 -11836.934,E2 -11836.934} C_VEL
LIN {X 0,Y 384.929,Z 396.965,A -85,B 0,C 180,E1 -11837.767,E2 -11837.767} C_VEL
LIN {X 0,Y 389.289,Z 421.482,A -85,B 0,C 180,E1 -11838.514,E2 -11838.514} C_VEL
LIN {X 0,Y 387.628,Z 505.898,A -85,B 0,C 180,E1 -11840.316,E2 -11840.316} C_VEL
LIN {X 0,Y 387.191,Z 518.462,A -85,B 0,C 180,E1 -11840.768,E2 -11840.768} C_VEL
LIN {X 0,Y 386.536,Z 532.042,A -85,B 0,C 180,E1 -11841.493,E2 -11841.493} C_VEL
LIN {X 0,Y 385.821,Z 544.534,A -85,B 0,C 180,E1 -11842.394,E2 -11842.394} C_VEL
LIN {X 0,Y 385.049,Z 556.381,A -85,B 0,C 180,E1 -11843.509,E2 -11843.509} C_VEL
LIN {X 0,Y 384.306,Z 566.289,A -85,B 0,C 180,E1 -11844.666,E2 -11844.666} C_VEL
LIN {X 0,Y 383.573,Z 575.711,A -85,B 0,C 180,E1 -11846.024,E2 -11846.024} C_VEL
LIN {X 0,Y 382.975,Z 584.418,A -85,B 0,C 180,E1 -11847.578,E2 -11847.578} C_VEL
LIN {X 0,Y 382.447,Z 591.038,A -85,B 0,C 180,E1 -11849.033,E2 -11849.033} C_VEL
LIN {X 0,Y 382.03,Z 597.458,A -85,B 0,C 180,E1 -11850.823,E2 -11850.823} C_VEL
LIN {X 0,Y 381.77,Z 602.292,A -85,B 0,C 180,E1 -11852.598,E2 -11852.598} C_VEL
LIN {X 0,Y 381.537,Z 605.958,A -85,B 0,C 180,E1 -11854.497,E2 -11854.497} C_VEL
LIN {X 0,Y 381.39,Z 607.909,A -85,B 0,C 180,E1 -11856.083,E2 -11856.083} C_VEL
LIN {X 0,Y 381.378,Z 608.696,A -85,B 0,C 180,E1 -11857.233,E2 -11857.233} C_VEL
LIN {X 0,Y 381.351,Z 609.03,A -85,B 0,C 180,E1 -11858.371,E2 -11858.371} C_VEL
LIN {X 0,Y 381.437,Z 608.631,A -85,B 0,C 180,E1 -11859.992,E2 -11859.992} C_VEL
LIN {X 0,Y 381.595,Z 607.083,A -85,B 0,C 180,E1 -11861.754,E2 -11861.754} C_VEL
LIN {X 0,Y 381.796,Z 604.955,A -85,B 0,C 180,E1 -11863.17,E2 -11863.17} C_VEL
LIN {X 0,Y 382.12,Z 600.805,A -85,B 0,C 180,E1 -11865.079,E2 -11865.079} C_VEL
LIN {X 0,Y 382.631,Z 595.771,A -85,B 0,C 180,E1 -11866.767,E2 -11866.767} C_VEL
LIN {X 0,Y 383.187,Z 589.715,A -85,B 0,C 180,E1 -11868.361,E2 -11868.361} C_VEL
LIN {X 0,Y 383.987,Z 581.942,A -85,B 0,C 180,E1 -11869.987,E2 -11869.987} C_VEL
LIN {X 0,Y 384.899,Z 573.425,A -85,B 0,C 180,E1 -11871.414,E2 -11871.414} C_VEL
LIN {X 0,Y 385.866,Z 563.199,A -85,B 0,C 180,E1 -11872.807,E2 -11872.807} C_VEL
LIN {X 0,Y 386.919,Z 552.051,A -85,B 0,C 180,E1 -11874.005,E2 -11874.005} C_VEL
LIN {X 0,Y 387.864,Z 539.985,A -85,B 0,C 180,E1 -11875.034,E2 -11875.034} C_VEL
LIN {X 0,Y 388.673,Z 527.301,A -85,B 0,C 180,E1 -11875.852,E2 -11875.852} C_VEL
LIN {X 0,Y 389.356,Z 514.053,A -85,B 0,C 180,E1 -11876.475,E2 -11876.475} C_VEL
LIN {X 0,Y 389.876,Z 499.515,A -85,B 0,C 180,E1 -11876.9,E2 -11876.9} C_VEL
LIN {X 0,Y 391.838,Z 422.033,A -85,B 0,C 180,E1 -11878.64,E2 -11878.64} C_VEL
LIN {X 0,Y 387.995,Z 404.136,A -85,B 0,C 180,E1 -11879.372,E2 -11879.372} C_VEL
LIN {X 0,Y 386.314,Z 397.991,A -85,B 0,C 180,E1 -11879.682,E2 -11879.682} C_VEL
LIN {X 0,Y 385.006,Z 390.977,A -85,B 0,C 180,E1 -11881.307,E2 -11881.307} C_VEL
LIN {X 0,Y 383.268,Z 383.748,A -85,B 0,C 180,E1 -11883.022,E2 -11883.022} C_VEL
LIN {X 0,Y 383.276,Z 383.745,A -85,B 0,C 180,E1 -11886.316,E2 -11886.316} C_VEL
LIN {X 0,Y 383.249,Z 383.746,A -85,B 0,C 180,E1 -11888.436,E2 -11888.436} C_VEL
LIN {X 0,Y 383.097,Z 383.767,A -85,B 0,C 180,E1 -11891.642,E2 -11891.642} C_VEL
LIN {X 0,Y 383.104,Z 383.765,A -85,B 0,C 180,E1 -11894.882,E2 -11894.882} C_VEL
LIN {X 0,Y 383.084,Z 383.768,A -85,B 0,C 180,E1 -11898.173,E2 -11898.173} C_VEL
LIN {X 0,Y 383.066,Z 383.768,A -85,B 0,C 180,E1 -11901.527,E2 -11901.527} C_VEL
LIN {X 0,Y 383.045,Z 383.77,A -85,B 0,C 180,E1 -11904.961,E2 -11904.961} C_VEL
LIN {X 0,Y 383.04,Z 383.771,A -85,B 0,C 180,E1 -11908.493,E2 -11908.493} C_VEL
LIN {X 0,Y 382.999,Z 383.776,A -85,B 0,C 180,E1 -11912.428,E2 -11912.428} C_VEL
LIN {X 0,Y 383.025,Z 383.773,A -85,B 0,C 180,E1 -11916.166,E2 -11916.166} C_VEL
LIN {X 0,Y 383.002,Z 383.776,A -85,B 0,C 180,E1 -11919.959,E2 -11919.959} C_VEL
LIN {X 0,Y 382.997,Z 383.776,A -85,B 0,C 180,E1 -11922.78,E2 -11922.78} C_VEL
LIN {X 0,Y 382.994,Z 383.776,A -85,B 0,C 180,E1 -11925.791,E2 -11925.791} C_VEL
LIN {X 0,Y 382.983,Z 383.78,A -85,B 0,C 180,E1 -11928.797,E2 -11928.797} C_VEL
LIN {X 0,Y 382.996,Z 383.776,A -85,B 0,C 180,E1 -11932.097,E2 -11932.097} C_VEL
LIN {X 0,Y 383.013,Z 383.776,A -85,B 0,C 180,E1 -11935.334,E2 -11935.334} C_VEL
LIN {X 0,Y 383.033,Z 383.771,A -85,B 0,C 180,E1 -11937.855,E2 -11937.855} C_VEL
LIN {X 0,Y 383.095,Z 383.852,A -85,B 0,C 180,E1 -11941.327,E2 -11941.327} C_VEL
LIN {X 0,Y 385.586,Z 396.166,A -85,B 0,C 180,E1 -11944.351,E2 -11944.351} C_VEL
LIN {X 0,Y 386.454,Z 401.343,A -85,B 0,C 180,E1 -11945.582,E2 -11945.582} C_VEL
LIN {X 0,Y 385.375,Z 414.7,A -85,B 0,C 180,E1 -11948.527,E2 -11948.527} C_VEL
LIN {X 0,Y 388.912,Z 434.302,A -85,B 0,C 180,E1 -11949.304,E2 -11949.304} C_VEL
LIN {X 0,Y 390.794,Z 449.391,A -85,B 0,C 180,E1 -11949.816,E2 -11949.816} C_VEL
LIN {X 0,Y 388.842,Z 528.122,A -85,B 0,C 180,E1 -11951.631,E2 -11951.631} C_VEL
LIN {X 0,Y 388.079,Z 541.458,A -85,B 0,C 180,E1 -11952.139,E2 -11952.139} C_VEL
LIN {X 0,Y 387.255,Z 554.106,A -85,B 0,C 180,E1 -11952.85,E2 -11952.85} C_VEL
LIN {X 0,Y 386.3,Z 566.246,A -85,B 0,C 180,E1 -11953.758,E2 -11953.758} C_VEL
LIN {X 0,Y 385.339,Z 577.197,A -85,B 0,C 180,E1 -11954.802,E2 -11954.802} C_VEL
LIN {X 0,Y 384.462,Z 587.789,A -85,B 0,C 180,E1 -11956.077,E2 -11956.077} C_VEL
LIN {X 0,Y 383.757,Z 596.364,A -85,B 0,C 180,E1 -11957.306,E2 -11957.306} C_VEL
LIN {X 0,Y 382.889,Z 605.396,A -85,B 0,C 180,E1 -11958.889,E2 -11958.889} C_VEL
LIN {X 0,Y 382.343,Z 612.639,A -85,B 0,C 180,E1 -11960.479,E2 -11960.479} C_VEL
LIN {X 0,Y 381.949,Z 618.416,A -85,B 0,C 180,E1 -11962.069,E2 -11962.069} C_VEL
LIN {X 0,Y 381.688,Z 623.476,A -85,B 0,C 180,E1 -11963.881,E2 -11963.881} C_VEL
LIN {X 0,Y 381.625,Z 627.287,A -85,B 0,C 180,E1 -11965.777,E2 -11965.777} C_VEL
LIN {X 0,Y 381.547,Z 628.804,A -85,B 0,C 180,E1 -11966.834,E2 -11966.834} C_VEL
LIN {X 0,Y 381.561,Z 629.862,A -85,B 0,C 180,E1 -11967.89,E2 -11967.89} C_VEL
LIN {X 0,Y 381.617,Z 630.523,A -85,B 0,C 180,E1 -11968.946,E2 -11968.946} C_VEL
LIN {X 0,Y 381.639,Z 630.79,A -85,B 0,C 180,E1 -11970.001,E2 -11970.001} C_VEL
LIN {X 0,Y 381.602,Z 630.651,A -85,B 0,C 180,E1 -11971.057,E2 -11971.057} C_VEL
LIN {X 0,Y 381.559,Z 630.073,A -85,B 0,C 180,E1 -11972.113,E2 -11972.113} C_VEL
LIN {X 0,Y 381.626,Z 627.729,A -85,B 0,C 180,E1 -11974.226,E2 -11974.226} C_VEL
LIN {X 0,Y 381.689,Z 624.171,A -85,B 0,C 180,E1 -11976.12,E2 -11976.12} C_VEL
LIN {X 0,Y 381.978,Z 619.336,A -85,B 0,C 180,E1 -11977.933,E2 -11977.933} C_VEL
LIN {X 0,Y 382.471,Z 612.826,A -85,B 0,C 180,E1 -11979.787,E2 -11979.787} C_VEL
LIN {X 0,Y 383.063,Z 605.715,A -85,B 0,C 180,E1 -11981.376,E2 -11981.376} C_VEL
LIN {X 0,Y 384.013,Z 596.835,A -85,B 0,C 180,E1 -11982.957,E2 -11982.957} C_VEL
LIN {X 0,Y 384.901,Z 586.638,A -85,B 0,C 180,E1 -11984.423,E2 -11984.423} C_VEL
LIN {X 0,Y 385.979,Z 575.192,A -85,B 0,C 180,E1 -11985.716,E2 -11985.716} C_VEL
LIN {X 0,Y 386.993,Z 563.536,A -85,B 0,C 180,E1 -11986.757,E2 -11986.757} C_VEL
LIN {X 0,Y 388.002,Z 551.18,A -85,B 0,C 180,E1 -11987.595,E2 -11987.595} C_VEL
LIN {X 0,Y 388.767,Z 538.287,A -85,B 0,C 180,E1 -11988.24,E2 -11988.24} C_VEL
LIN {X 0,Y 389.39,Z 525.898,A -85,B 0,C 180,E1 -11988.652,E2 -11988.652} C_VEL
LIN {X 0,Y 390.709,Z 448.695,A -85,B 0,C 180,E1 -11990.183,E2 -11990.183} C_VEL
LIN {X 0,Y 387.043,Z 426.134,A -85,B 0,C 180,E1 -11990.877,E2 -11990.877} C_VEL
LIN {X 0,Y 385.483,Z 417.794,A -85,B 0,C 180,E1 -11991.182,E2 -11991.182} C_VEL
LIN {X 0,Y 386.759,Z 404.589,A -85,B 0,C 180,E1 -11994.134,E2 -11994.134} C_VEL
LIN {X 0,Y 386.8,Z 402.139,A -85,B 0,C 180,E1 -11994.703,E2 -11994.703} C_VEL
LIN {X 0,Y 384.732,Z 391.154,A -85,B 0,C 180,E1 -11997.469,E2 -11997.469} C_VEL
LIN {X 0,Y 383.045,Z 383.779,A -85,B 0,C 180,E1 -11999.47,E2 -11999.47} C_VEL
LIN {X 0,Y 383.008,Z 383.779,A -85,B 0,C 180,E1 -12003.402,E2 -12003.402} C_VEL
LIN {X 0,Y 383.037,Z 383.774,A -85,B 0,C 180,E1 -12006.165,E2 -12006.165} C_VEL
LIN {X 0,Y 383.014,Z 383.777,A -85,B 0,C 180,E1 -12009.959,E2 -12009.959} C_VEL
LIN {X 0,Y 383.011,Z 383.778,A -85,B 0,C 180,E1 -12012.779,E2 -12012.779} C_VEL
LIN {X 0,Y 383.003,Z 383.777,A -85,B 0,C 180,E1 -12015.79,E2 -12015.79} C_VEL
LIN {X 0,Y 382.994,Z 383.78,A -85,B 0,C 180,E1 -12018.796,E2 -12018.796} C_VEL
LIN {X 0,Y 383.004,Z 383.775,A -85,B 0,C 180,E1 -12022.097,E2 -12022.097} C_VEL
LIN {X 0,Y 383.024,Z 383.77,A -85,B 0,C 180,E1 -12025.333,E2 -12025.333} C_VEL
LIN {X 0,Y 382.989,Z 383.772,A -85,B 0,C 180,E1 -12029.082,E2 -12029.082} C_VEL
LIN {X 0,Y 383.062,Z 383.765,A -85,B 0,C 180,E1 -12032.699,E2 -12032.699} C_VEL
LIN {X 0,Y 383.057,Z 383.77,A -85,B 0,C 180,E1 -12035.04,E2 -12035.04} C_VEL
LIN {X 0,Y 383.005,Z 383.774,A -85,B 0,C 180,E1 -12038.47,E2 -12038.47} C_VEL
LIN {X 0,Y 383.069,Z 383.76,A -85,B 0,C 180,E1 -12041.827,E2 -12041.827} C_VEL
LIN {X 0,Y 383.116,Z 383.753,A -85,B 0,C 180,E1 -12045.119,E2 -12045.119} C_VEL
LIN {X 0,Y 383.104,Z 383.762,A -85,B 0,C 180,E1 -12048.358,E2 -12048.358} C_VEL
LIN {X 0,Y 383.31,Z 383.74,A -85,B 0,C 180,E1 -12051.933,E2 -12051.933} C_VEL
LIN {X 0,Y 383.205,Z 383.751,A -85,B 0,C 180,E1 -12054.739,E2 -12054.739} C_VEL
LIN {X 0,Y 383.392,Z 383.724,A -85,B 0,C 180,E1 -12057.899,E2 -12057.899} C_VEL
LIN {X 0,Y 383.524,Z 383.71,A -85,B 0,C 180,E1 -12060,E2 -12060} C_VEL
LIN {X 0,Y 383.253,Z 383.743,A -85,B 0,C 180,E1 -12063.154,E2 -12063.154} C_VEL
LIN {X 0,Y 383.276,Z 383.738,A -85,B 0,C 180,E1 -12066.63,E2 -12066.63} C_VEL
LIN {X 0,Y 383.267,Z 383.744,A -85,B 0,C 180,E1 -12068.436,E2 -12068.436} C_VEL
LIN {X 0,Y 383.104,Z 383.765,A -85,B 0,C 180,E1 -12071.642,E2 -12071.642} C_VEL
LIN {X 0,Y 383.117,Z 383.761,A -85,B 0,C 180,E1 -12074.882,E2 -12074.882} C_VEL
LIN {X 0,Y 383.096,Z 383.768,A -85,B 0,C 180,E1 -12078.172,E2 -12078.172} C_VEL
LIN {X 0,Y 382.999,Z 383.781,A -85,B 0,C 180,E1 -12081.531,E2 -12081.531} C_VEL
LIN {X 0,Y 383.058,Z 383.772,A -85,B 0,C 180,E1 -12084.96,E2 -12084.96} C_VEL
LIN {X 0,Y 383.103,Z 383.895,A -85,B 0,C 180,E1 -12086.488,E2 -12086.488} C_VEL
LIN {X 0,Y 385.251,Z 394.213,A -85,B 0,C 180,E1 -12089.509,E2 -12089.509} C_VEL
LIN {X 0,Y 385.959,Z 399.532,A -85,B 0,C 180,E1 -12090.947,E2 -12090.947} C_VEL
LIN {X 0,Y 389.91,Z 416.387,A -85,B 0,C 180,E1 -12091.553,E2 -12091.553} C_VEL
LIN {X 0,Y 391.085,Z 422.387,A -85,B 0,C 180,E1 -12091.75,E2 -12091.75} C_VEL
LIN {X 0,Y 389.497,Z 506.723,A -85,B 0,C 180,E1 -12093.429,E2 -12093.429} C_VEL
LIN {X 0,Y 388.962,Z 520.127,A -85,B 0,C 180,E1 -12093.911,E2 -12093.911} C_VEL
LIN {X 0,Y 388.318,Z 531.773,A -85,B 0,C 180,E1 -12094.522,E2 -12094.522} C_VEL
LIN {X 0,Y 387.473,Z 544.136,A -85,B 0,C 180,E1 -12095.399,E2 -12095.399} C_VEL
LIN {X 0,Y 386.455,Z 556.098,A -85,B 0,C 180,E1 -12096.502,E2 -12096.502} C_VEL
LIN {X 0,Y 385.588,Z 565.86,A -85,B 0,C 180,E1 -12097.633,E2 -12097.633} C_VEL
LIN {X 0,Y 384.498,Z 575.894,A -85,B 0,C 180,E1 -12099.078,E2 -12099.078} C_VEL
LIN {X 0,Y 383.666,Z 584.149,A -85,B 0,C 180,E1 -12100.554,E2 -12100.554} C_VEL
LIN {X 0,Y 383.038,Z 590.772,A -85,B 0,C 180,E1 -12102.013,E2 -12102.013} C_VEL
LIN {X 0,Y 382.437,Z 597.384,A -85,B 0,C 180,E1 -12103.854,E2 -12103.854} C_VEL
LIN {X 0,Y 381.949,Z 602.75,A -85,B 0,C 180,E1 -12105.858,E2 -12105.858} C_VEL
LIN {X 0,Y 381.664,Z 605.783,A -85,B 0,C 180,E1 -12107.44,E2 -12107.44} C_VEL
LIN {X 0,Y 381.501,Z 607.876,A -85,B 0,C 180,E1 -12109.052,E2 -12109.052} C_VEL
LIN {X 0,Y 381.361,Z 609.198,A -85,B 0,C 180,E1 -12111.201,E2 -12111.201} C_VEL
LIN {X 0,Y 381.357,Z 609.176,A -85,B 0,C 180,E1 -12112.543,E2 -12112.543} C_VEL
LIN {X 0,Y 381.399,Z 608.273,A -85,B 0,C 180,E1 -12114.173,E2 -12114.173} C_VEL
LIN {X 0,Y 381.541,Z 606.146,A -85,B 0,C 180,E1 -12115.987,E2 -12115.987} C_VEL
LIN {X 0,Y 381.881,Z 602.637,A -85,B 0,C 180,E1 -12117.841,E2 -12117.841} C_VEL
LIN {X 0,Y 382.23,Z 597.386,A -85,B 0,C 180,E1 -12119.79,E2 -12119.79} C_VEL
LIN {X 0,Y 382.744,Z 591.375,A -85,B 0,C 180,E1 -12121.482,E2 -12121.482} C_VEL
LIN {X 0,Y 383.317,Z 584.524,A -85,B 0,C 180,E1 -12123.012,E2 -12123.012} C_VEL
LIN {X 0,Y 384.036,Z 576.095,A -85,B 0,C 180,E1 -12124.527,E2 -12124.527} C_VEL
LIN {X 0,Y 384.883,Z 566.498,A -85,B 0,C 180,E1 -12125.925,E2 -12125.925} C_VEL
LIN {X 0,Y 385.749,Z 556.69,A -85,B 0,C 180,E1 -12127.08,E2 -12127.08} C_VEL
LIN {X 0,Y 386.567,Z 545.433,A -85,B 0,C 180,E1 -12128.139,E2 -12128.139} C_VEL
LIN {X 0,Y 387.381,Z 532.674,A -85,B 0,C 180,E1 -12129.072,E2 -12129.072} C_VEL
LIN {X 0,Y 387.997,Z 520.432,A -85,B 0,C 180,E1 -12129.73,E2 -12129.73} C_VEL
LIN {X 0,Y 388.533,Z 507.069,A -85,B 0,C 180,E1 -12130.216,E2 -12130.216} C_VEL
LIN {X 0,Y 389.126,Z 474.479,A -85,B 0,C 180,E1 -12130.881,E2 -12130.881} C_VEL
LIN {X 0,Y 389.865,Z 421.537,A -85,B 0,C 180,E1 -12131.907,E2 -12131.907} C_VEL
LIN {X 0,Y 385.345,Z 398.441,A -85,B 0,C 180,E1 -12132.622,E2 -12132.622} C_VEL
LIN {X 0,Y 385.155,Z 394.798,A -85,B 0,C 180,E1 -12133.569,E2 -12133.569} C_VEL
LIN {X 0,Y 383.155,Z 383.76,A -85,B 0,C 180,E1 -12136.588,E2 -12136.588} C_VEL
LIN {X 0,Y 383.152,Z 383.759,A -85,B 0,C 180,E1 -12140.629,E2 -12140.629} C_VEL
LIN {X 0,Y 383.26,Z 383.741,A -85,B 0,C 180,E1 -12143.682,E2 -12143.682} C_VEL
LIN {X 0,Y 383.125,Z 383.758,A -85,B 0,C 180,E1 -12145.204,E2 -12145.204} C_VEL
LIN {X 0,Y 382.399,Z 383.853,A -85,B 0,C 180,E1 -12146.082,E2 -12146.082} C_VEL
LIN {X 0,Y 379.584,Z 384.199,A -85,B 0,C 180,E1 -12147.513,E2 -12147.513} C_VEL
LIN {X 0,Y 377.324,Z 384.483,A -85,B 0,C 180,E1 -12148.67,E2 -12148.67} C_VEL
LIN {X 0,Y 376.469,Z 384.587,A -85,B 0,C 180,E1 -12149.563,E2 -12149.563} C_VEL
LIN {X 0,Y 376.458,Z 384.59,A -85,B 0,C 180,E1 -12149.864,E2 -12149.864} C_VEL
LIN {X 0,Y 376.357,Z 384.605,A -85,B 0,C 180,E1 -12152.139,E2 -12152.139} C_VEL
LIN {X 0,Y 376.25,Z 384.618,A -85,B 0,C 180,E1 -12156.433,E2 -12156.433} C_VEL
LIN {X 0,Y 376.207,Z 384.622,A -85,B 0,C 180,E1 -12158.594,E2 -12158.594} C_VEL
LIN {X 0,Y 376.051,Z 384.643,A -85,B 0,C 180,E1 -12161.862,E2 -12161.862} C_VEL
LIN {X 0,Y 376.062,Z 384.637,A -85,B 0,C 180,E1 -12165.166,E2 -12165.166} C_VEL
LIN {X 0,Y 376.024,Z 384.643,A -85,B 0,C 180,E1 -12168.524,E2 -12168.524} C_VEL
LIN {X 0,Y 375.956,Z 384.657,A -85,B 0,C 180,E1 -12171.953,E2 -12171.953} C_VEL
LIN {X 0,Y 376.004,Z 384.647,A -85,B 0,C 180,E1 -12175.459,E2 -12175.459} C_VEL
LIN {X 0,Y 375.979,Z 384.648,A -85,B 0,C 180,E1 -12179.077,E2 -12179.077} C_VEL
LIN {X 0,Y 375.955,Z 384.651,A -85,B 0,C 180,E1 -12182.826,E2 -12182.826} C_VEL
LIN {X 0,Y 375.954,Z 384.655,A -85,B 0,C 180,E1 -12185.414,E2 -12185.414} C_VEL
LIN {X 0,Y 375.973,Z 384.649,A -85,B 0,C 180,E1 -12188.27,E2 -12188.27} C_VEL
LIN {X 0,Y 375.956,Z 384.657,A -85,B 0,C 180,E1 -12191.604,E2 -12191.604} C_VEL
LIN {X 0,Y 376.026,Z 384.73,A -85,B 0,C 180,E1 -12194.651,E2 -12194.651} C_VEL
LIN {X 0,Y 377.84,Z 394.544,A -85,B 0,C 180,E1 -12196.889,E2 -12196.889} C_VEL
LIN {X 0,Y 377.99,Z 397.093,A -85,B 0,C 180,E1 -12197.453,E2 -12197.453} C_VEL
LIN {X 0,Y 382.457,Z 422.295,A -85,B 0,C 180,E1 -12198.239,E2 -12198.239} C_VEL
LIN {X 0,Y 380.713,Z 506.578,A -85,B 0,C 180,E1 -12200.084,E2 -12200.084} C_VEL
LIN {X 0,Y 380.267,Z 518.843,A -85,B 0,C 180,E1 -12200.539,E2 -12200.539} C_VEL
LIN {X 0,Y 379.627,Z 531.872,A -85,B 0,C 180,E1 -12201.246,E2 -12201.246} C_VEL
LIN {X 0,Y 378.958,Z 543.628,A -85,B 0,C 180,E1 -12202.097,E2 -12202.097} C_VEL
LIN {X 0,Y 378.182,Z 554.722,A -85,B 0,C 180,E1 -12203.124,E2 -12203.124} C_VEL
LIN {X 0,Y 377.374,Z 565.777,A -85,B 0,C 180,E1 -12204.41,E2 -12204.41} C_VEL
LIN {X 0,Y 376.67,Z 574.638,A -85,B 0,C 180,E1 -12205.675,E2 -12205.675} C_VEL
LIN {X 0,Y 375.971,Z 583.603,A -85,B 0,C 180,E1 -12207.262,E2 -12207.262} C_VEL
LIN {X 0,Y 375.377,Z 591.41,A -85,B 0,C 180,E1 -12208.987,E2 -12208.987} C_VEL
LIN {X 0,Y 374.93,Z 597.857,A -85,B 0,C 180,E1 -12210.832,E2 -12210.832} C_VEL
LIN {X 0,Y 374.673,Z 602.651,A -85,B 0,C 180,E1 -12212.641,E2 -12212.641} C_VEL
LIN {X 0,Y 374.469,Z 606.042,A -85,B 0,C 180,E1 -12214.427,E2 -12214.427} C_VEL
LIN {X 0,Y 374.316,Z 607.566,A -85,B 0,C 180,E1 -12215.602,E2 -12215.602} C_VEL
LIN {X 0,Y 374.274,Z 608.723,A -85,B 0,C 180,E1 -12216.937,E2 -12216.937} C_VEL
LIN {X 0,Y 374.267,Z 609.134,A -85,B 0,C 180,E1 -12217.941,E2 -12217.941} C_VEL
LIN {X 0,Y 374.349,Z 608.938,A -85,B 0,C 180,E1 -12219.828,E2 -12219.828} C_VEL
LIN {X 0,Y 374.45,Z 607.804,A -85,B 0,C 180,E1 -12221.393,E2 -12221.393} C_VEL
LIN {X 0,Y 374.698,Z 605.624,A -85,B 0,C 180,E1 -12223.047,E2 -12223.047} C_VEL
LIN {X 0,Y 374.983,Z 602.2,A -85,B 0,C 180,E1 -12224.788,E2 -12224.788} C_VEL
LIN {X 0,Y 375.535,Z 597.01,A -85,B 0,C 180,E1 -12226.687,E2 -12226.687} C_VEL
LIN {X 0,Y 376.155,Z 590.762,A -85,B 0,C 180,E1 -12228.413,E2 -12228.413} C_VEL
LIN {X 0,Y 376.985,Z 583.193,A -85,B 0,C 180,E1 -12230.07,E2 -12230.07} C_VEL
LIN {X 0,Y 377.838,Z 575.45,A -85,B 0,C 180,E1 -12231.442,E2 -12231.442} C_VEL
LIN {X 0,Y 378.936,Z 564.935,A -85,B 0,C 180,E1 -12232.942,E2 -12232.942} C_VEL
LIN {X 0,Y 380.051,Z 554.27,A -85,B 0,C 180,E1 -12234.162,E2 -12234.162} C_VEL
LIN {X 0,Y 381.035,Z 542.887,A -85,B 0,C 180,E1 -12235.195,E2 -12235.195} C_VEL
LIN {X 0,Y 381.95,Z 529.899,A -85,B 0,C 180,E1 -12236.109,E2 -12236.109} C_VEL
LIN {X 0,Y 382.688,Z 516.733,A -85,B 0,C 180,E1 -12236.776,E2 -12236.776} C_VEL
LIN {X 0,Y 383.201,Z 504.153,A -85,B 0,C 180,E1 -12237.208,E2 -12237.208} C_VEL
LIN {X 0,Y 385.479,Z 423.442,A -85,B 0,C 180,E1 -12239.063,E2 -12239.063} C_VEL
LIN {X 0,Y 382.029,Z 406.997,A -85,B 0,C 180,E1 -12239.765,E2 -12239.765} C_VEL
LIN {X 0,Y 379.875,Z 399.853,A -85,B 0,C 180,E1 -12240.128,E2 -12240.128} C_VEL
LIN {X 0,Y 379.338,Z 398.239,A -85,B 0,C 180,E1 -12240.219,E2 -12240.219} C_VEL
LIN {X 0,Y 377.123,Z 387.985,A -85,B 0,C 180,E1 -12242.67,E2 -12242.67} C_VEL
LIN {X 0,Y 376.135,Z 384.637,A -85,B 0,C 180,E1 -12243.548,E2 -12243.548} C_VEL
LIN {X 0,Y 376.236,Z 384.621,A -85,B 0,C 180,E1 -12246.435,E2 -12246.435} C_VEL
LIN {X 0,Y 376.195,Z 384.625,A -85,B 0,C 180,E1 -12248.595,E2 -12248.595} C_VEL
LIN {X 0,Y 376.048,Z 384.643,A -85,B 0,C 180,E1 -12251.863,E2 -12251.863} C_VEL
LIN {X 0,Y 376.052,Z 384.643,A -85,B 0,C 180,E1 -12255.168,E2 -12255.168} C_VEL
LIN {X 0,Y 376.021,Z 384.648,A -85,B 0,C 180,E1 -12258.526,E2 -12258.526} C_VEL
LIN {X 0,Y 376.015,Z 384.65,A -85,B 0,C 180,E1 -12261.951,E2 -12261.951} C_VEL
LIN {X 0,Y 375.998,Z 384.65,A -85,B 0,C 180,E1 -12265.462,E2 -12265.462} C_VEL
LIN {X 0,Y 375.967,Z 384.653,A -85,B 0,C 180,E1 -12269.079,E2 -12269.079} C_VEL
LIN {X 0,Y 375.949,Z 384.654,A -85,B 0,C 180,E1 -12272.829,E2 -12272.829} C_VEL
LIN {X 0,Y 375.949,Z 384.655,A -85,B 0,C 180,E1 -12275.416,E2 -12275.416} C_VEL
LIN {X 0,Y 375.968,Z 384.652,A -85,B 0,C 180,E1 -12278.272,E2 -12278.272} C_VEL
LIN {X 0,Y 375.928,Z 384.659,A -85,B 0,C 180,E1 -12281.602,E2 -12281.602} C_VEL
LIN {X 0,Y 375.948,Z 384.657,A -85,B 0,C 180,E1 -12285.265,E2 -12285.265} C_VEL
LIN {X 0,Y 375.935,Z 384.657,A -85,B 0,C 180,E1 -12289.134,E2 -12289.134} C_VEL
LIN {X 0,Y 375.96,Z 384.652,A -85,B 0,C 180,E1 -12291.913,E2 -12291.913} C_VEL
LIN {X 0,Y 375.975,Z 384.653,A -85,B 0,C 180,E1 -12295.334,E2 -12295.334} C_VEL
LIN {X 0,Y 375.973,Z 384.653,A -85,B 0,C 180,E1 -12298.441,E2 -12298.441} C_VEL
LIN {X 0,Y 376.043,Z 384.73,A -85,B 0,C 180,E1 -12301.039,E2 -12301.039} C_VEL
LIN {X 0,Y 378.314,Z 395.79,A -85,B 0,C 180,E1 -12303.821,E2 -12303.821} C_VEL
LIN {X 0,Y 379.503,Z 403.094,A -85,B 0,C 180,E1 -12305.587,E2 -12305.587} C_VEL
LIN {X 0,Y 378.586,Z 413.936,A -85,B 0,C 180,E1 -12307.98,E2 -12307.98} C_VEL
LIN {X 0,Y 382.33,Z 434.054,A -85,B 0,C 180,E1 -12308.811,E2 -12308.811} C_VEL
LIN {X 0,Y 384.36,Z 450.549,A -85,B 0,C 180,E1 -12309.393,E2 -12309.393} C_VEL
LIN {X 0,Y 382.279,Z 528.124,A -85,B 0,C 180,E1 -12311.234,E2 -12311.234} C_VEL
LIN {X 0,Y 381.454,Z 541.37,A -85,B 0,C 180,E1 -12311.749,E2 -12311.749} C_VEL
LIN {X 0,Y 380.676,Z 553,A -85,B 0,C 180,E1 -12312.405,E2 -12312.405} C_VEL
LIN {X 0,Y 379.642,Z 565.306,A -85,B 0,C 180,E1 -12313.327,E2 -12313.327} C_VEL
LIN {X 0,Y 378.62,Z 576.394,A -85,B 0,C 180,E1 -12314.388,E2 -12314.388} C_VEL
LIN {X 0,Y 377.759,Z 585.936,A -85,B 0,C 180,E1 -12315.529,E2 -12315.529} C_VEL
LIN {X 0,Y 376.984,Z 594.673,A -85,B 0,C 180,E1 -12316.8,E2 -12316.8} C_VEL
LIN {X 0,Y 376.001,Z 603.741,A -85,B 0,C 180,E1 -12318.41,E2 -12318.41} C_VEL
LIN {X 0,Y 375.293,Z 612.291,A -85,B 0,C 180,E1 -12320.299,E2 -12320.299} C_VEL
LIN {X 0,Y 374.887,Z 618.102,A -85,B 0,C 180,E1 -12321.919,E2 -12321.919} C_VEL
LIN {X 0,Y 374.629,Z 622.67,A -85,B 0,C 180,E1 -12323.539,E2 -12323.539} C_VEL
LIN {X 0,Y 374.553,Z 625.069,A -85,B 0,C 180,E1 -12324.618,E2 -12324.618} C_VEL
LIN {X 0,Y 374.551,Z 627.032,A -85,B 0,C 180,E1 -12325.697,E2 -12325.697} C_VEL
LIN {X 0,Y 374.462,Z 628.564,A -85,B 0,C 180,E1 -12326.774,E2 -12326.774} C_VEL
LIN {X 0,Y 374.46,Z 629.637,A -85,B 0,C 180,E1 -12327.85,E2 -12327.85} C_VEL
LIN {X 0,Y 374.517,Z 630.307,A -85,B 0,C 180,E1 -12328.926,E2 -12328.926} C_VEL
LIN {X 0,Y 374.553,Z 630.584,A -85,B 0,C 180,E1 -12330.001,E2 -12330.001} C_VEL
LIN {X 0,Y 374.502,Z 630.459,A -85,B 0,C 180,E1 -12331.077,E2 -12331.077} C_VEL
LIN {X 0,Y 374.458,Z 629.892,A -85,B 0,C 180,E1 -12332.153,E2 -12332.153} C_VEL
LIN {X 0,Y 374.53,Z 627.563,A -85,B 0,C 180,E1 -12334.306,E2 -12334.306} C_VEL
LIN {X 0,Y 374.584,Z 624.393,A -85,B 0,C 180,E1 -12336.068,E2 -12336.068} C_VEL
LIN {X 0,Y 374.804,Z 620.765,A -85,B 0,C 180,E1 -12337.544,E2 -12337.544} C_VEL
LIN {X 0,Y 375.195,Z 615.713,A -85,B 0,C 180,E1 -12339.163,E2 -12339.163} C_VEL
LIN {X 0,Y 375.738,Z 609.373,A -85,B 0,C 180,E1 -12340.782,E2 -12340.782} C_VEL
LIN {X 0,Y 376.578,Z 601.445,A -85,B 0,C 180,E1 -12342.395,E2 -12342.395} C_VEL
LIN {X 0,Y 377.595,Z 591.587,A -85,B 0,C 180,E1 -12344.004,E2 -12344.004} C_VEL
LIN {X 0,Y 378.446,Z 582.493,A -85,B 0,C 180,E1 -12345.209,E2 -12345.209} C_VEL
LIN {X 0,Y 379.538,Z 571.246,A -85,B 0,C 180,E1 -12346.404,E2 -12346.404} C_VEL
LIN {X 0,Y 380.551,Z 560.26,A -85,B 0,C 180,E1 -12347.327,E2 -12347.327} C_VEL
LIN {X 0,Y 381.438,Z 548.156,A -85,B 0,C 180,E1 -12348.116,E2 -12348.116} C_VEL
LIN {X 0,Y 382.22,Z 535.668,A -85,B 0,C 180,E1 -12348.702,E2 -12348.702} C_VEL
LIN {X 0,Y 382.842,Z 522.87,A -85,B 0,C 180,E1 -12349.088,E2 -12349.088} C_VEL
LIN {X 0,Y 384.062,Z 449.139,A -85,B 0,C 180,E1 -12350.574,E2 -12350.574} C_VEL
LIN {X 0,Y 380.267,Z 425.712,A -85,B 0,C 180,E1 -12351.316,E2 -12351.316} C_VEL
LIN {X 0,Y 378.683,Z 417.687,A -85,B 0,C 180,E1 -12351.603,E2 -12351.603} C_VEL
LIN {X 0,Y 379.926,Z 405.101,A -85,B 0,C 180,E1 -12354.482,E2 -12354.482} C_VEL
LIN {X 0,Y 379.222,Z 399.723,A -85,B 0,C 180,E1 -12355.82,E2 -12355.82} C_VEL
LIN {X 0,Y 376.893,Z 388.478,A -85,B 0,C 180,E1 -12358.786,E2 -12358.786} C_VEL
LIN {X 0,Y 375.982,Z 384.657,A -85,B 0,C 180,E1 -12359.848,E2 -12359.848} C_VEL
LIN {X 0,Y 375.954,Z 384.657,A -85,B 0,C 180,E1 -12362.829,E2 -12362.829} C_VEL
LIN {X 0,Y 375.963,Z 384.655,A -85,B 0,C 180,E1 -12365.416,E2 -12365.416} C_VEL
LIN {X 0,Y 375.98,Z 384.654,A -85,B 0,C 180,E1 -12368.271,E2 -12368.271} C_VEL
LIN {X 0,Y 375.94,Z 384.66,A -85,B 0,C 180,E1 -12371.602,E2 -12371.602} C_VEL
LIN {X 0,Y 375.932,Z 384.66,A -85,B 0,C 180,E1 -12375.269,E2 -12375.269} C_VEL
LIN {X 0,Y 375.94,Z 384.656,A -85,B 0,C 180,E1 -12378.4,E2 -12378.4} C_VEL
LIN {X 0,Y 375.978,Z 384.65,A -85,B 0,C 180,E1 -12381.73,E2 -12381.73} C_VEL
LIN {X 0,Y 375.985,Z 384.646,A -85,B 0,C 180,E1 -12385.333,E2 -12385.333} C_VEL
LIN {X 0,Y 375.964,Z 384.655,A -85,B 0,C 180,E1 -12388.439,E2 -12388.439} C_VEL
LIN {X 0,Y 375.989,Z 384.649,A -85,B 0,C 180,E1 -12392.141,E2 -12392.141} C_VEL
LIN {X 0,Y 376.012,Z 384.645,A -85,B 0,C 180,E1 -12394.539,E2 -12394.539} C_VEL
LIN {X 0,Y 375.974,Z 384.646,A -85,B 0,C 180,E1 -12398.046,E2 -12398.046} C_VEL
LIN {X 0,Y 376.015,Z 384.637,A -85,B 0,C 180,E1 -12401.474,E2 -12401.474} C_VEL
LIN {X 0,Y 376.065,Z 384.633,A -85,B 0,C 180,E1 -12404.833,E2 -12404.833} C_VEL
LIN {X 0,Y 376.056,Z 384.643,A -85,B 0,C 180,E1 -12408.137,E2 -12408.137} C_VEL
LIN {X 0,Y 376.264,Z 384.617,A -85,B 0,C 180,E1 -12411.878,E2 -12411.878} C_VEL
LIN {X 0,Y 376.177,Z 384.627,A -85,B 0,C 180,E1 -12414.64,E2 -12414.64} C_VEL
LIN {X 0,Y 376.358,Z 384.599,A -85,B 0,C 180,E1 -12417.86,E2 -12417.86} C_VEL
LIN {X 0,Y 376.493,Z 384.585,A -85,B 0,C 180,E1 -12420,E2 -12420} C_VEL
LIN {X 0,Y 376.191,Z 384.623,A -85,B 0,C 180,E1 -12423.213,E2 -12423.213} C_VEL
LIN {X 0,Y 376.241,Z 384.614,A -85,B 0,C 180,E1 -12426.621,E2 -12426.621} C_VEL
LIN {X 0,Y 376.212,Z 384.622,A -85,B 0,C 180,E1 -12428.595,E2 -12428.595} C_VEL
LIN {X 0,Y 376.056,Z 384.642,A -85,B 0,C 180,E1 -12431.863,E2 -12431.863} C_VEL
LIN {X 0,Y 376.065,Z 384.641,A -85,B 0,C 180,E1 -12435.167,E2 -12435.167} C_VEL
LIN {X 0,Y 376.03,Z 384.646,A -85,B 0,C 180,E1 -12438.526,E2 -12438.526} C_VEL
LIN {X 0,Y 375.97,Z 384.654,A -85,B 0,C 180,E1 -12441.954,E2 -12441.954} C_VEL
LIN {X 0,Y 376.016,Z 384.646,A -85,B 0,C 180,E1 -12445.461,E2 -12445.461} C_VEL
LIN {X 0,Y 376.087,Z 384.809,A -85,B 0,C 180,E1 -12446.109,E2 -12446.109} C_VEL
LIN {X 0,Y 378.207,Z 394.928,A -85,B 0,C 180,E1 -12449.145,E2 -12449.145} C_VEL
LIN {X 0,Y 378.95,Z 399.543,A -85,B 0,C 180,E1 -12450.472,E2 -12450.472} C_VEL
LIN {X 0,Y 381.821,Z 410.188,A -85,B 0,C 180,E1 -12450.908,E2 -12450.908} C_VEL
LIN {X 0,Y 384.554,Z 423.882,A -85,B 0,C 180,E1 -12451.378,E2 -12451.378} C_VEL
LIN {X 0,Y 382.864,Z 506.847,A -85,B 0,C 180,E1 -12453.058,E2 -12453.058} C_VEL
LIN {X 0,Y 382.287,Z 520.497,A -85,B 0,C 180,E1 -12453.557,E2 -12453.557} C_VEL
LIN {X 0,Y 381.643,Z 531.853,A -85,B 0,C 180,E1 -12454.164,E2 -12454.164} C_VEL
LIN {X 0,Y 380.73,Z 544.347,A -85,B 0,C 180,E1 -12455.062,E2 -12455.062} C_VEL
LIN {X 0,Y 379.724,Z 555.728,A -85,B 0,C 180,E1 -12456.124,E2 -12456.124} C_VEL
LIN {X 0,Y 378.712,Z 566.526,A -85,B 0,C 180,E1 -12457.396,E2 -12457.396} C_VEL
LIN {X 0,Y 377.762,Z 574.911,A -85,B 0,C 180,E1 -12458.611,E2 -12458.611} C_VEL
LIN {X 0,Y 376.823,Z 583.393,A -85,B 0,C 180,E1 -12460.12,E2 -12460.12} C_VEL
LIN {X 0,Y 376.143,Z 590.299,A -85,B 0,C 180,E1 -12461.635,E2 -12461.635} C_VEL
LIN {X 0,Y 375.603,Z 595.856,A -85,B 0,C 180,E1 -12463.134,E2 -12463.134} C_VEL
LIN {X 0,Y 375.04,Z 601.428,A -85,B 0,C 180,E1 -12465.053,E2 -12465.053} C_VEL
LIN {X 0,Y 374.647,Z 605.488,A -85,B 0,C 180,E1 -12467.021,E2 -12467.021} C_VEL
LIN {X 0,Y 374.415,Z 608.042,A -85,B 0,C 180,E1 -12468.929,E2 -12468.929} C_VEL
LIN {X 0,Y 374.308,Z 609.102,A -85,B 0,C 180,E1 -12470.338,E2 -12470.338} C_VEL
LIN {X 0,Y 374.246,Z 609.454,A -85,B 0,C 180,E1 -12472.067,E2 -12472.067} C_VEL
LIN {X 0,Y 374.28,Z 608.731,A -85,B 0,C 180,E1 -12473.846,E2 -12473.846} C_VEL
LIN {X 0,Y 374.422,Z 606.757,A -85,B 0,C 180,E1 -12475.728,E2 -12475.728} C_VEL
LIN {X 0,Y 374.734,Z 603.595,A -85,B 0,C 180,E1 -12477.561,E2 -12477.561} C_VEL
LIN {X 0,Y 375.09,Z 598.473,A -85,B 0,C 180,E1 -12479.608,E2 -12479.608} C_VEL
LIN {X 0,Y 375.574,Z 592.957,A -85,B 0,C 180,E1 -12481.258,E2 -12481.258} C_VEL
LIN {X 0,Y 376.265,Z 585.29,A -85,B 0,C 180,E1 -12483.066,E2 -12483.066} C_VEL
LIN {X 0,Y 376.995,Z 577.001,A -85,B 0,C 180,E1 -12484.609,E2 -12484.609} C_VEL
LIN {X 0,Y 377.934,Z 566.738,A -85,B 0,C 180,E1 -12486.141,E2 -12486.141} C_VEL
LIN {X 0,Y 378.953,Z 555.93,A -85,B 0,C 180,E1 -12487.42,E2 -12487.42} C_VEL
LIN {X 0,Y 379.709,Z 545.459,A -85,B 0,C 180,E1 -12488.415,E2 -12488.415} C_VEL
LIN {X 0,Y 380.507,Z 533.413,A -85,B 0,C 180,E1 -12489.313,E2 -12489.313} C_VEL
LIN {X 0,Y 381.2,Z 520.464,A -85,B 0,C 180,E1 -12490.026,E2 -12490.026} C_VEL
LIN {X 0,Y 381.749,Z 506.585,A -85,B 0,C 180,E1 -12490.535,E2 -12490.535} C_VEL
LIN {X 0,Y 383.196,Z 422.796,A -85,B 0,C 180,E1 -12492.211,E2 -12492.211} C_VEL
LIN {X 0,Y 378.427,Z 398.58,A -85,B 0,C 180,E1 -12492.991,E2 -12492.991} C_VEL
LIN {X 0,Y 377.42,Z 391.619,A -85,B 0,C 180,E1 -12494.887,E2 -12494.887} C_VEL
LIN {X 0,Y 376.087,Z 384.641,A -85,B 0,C 180,E1 -12496.843,E2 -12496.843} C_VEL
LIN {X 0,Y 376.124,Z 384.634,A -85,B 0,C 180,E1 -12500.317,E2 -12500.317} C_VEL
LIN {X 0,Y 376.218,Z 384.618,A -85,B 0,C 180,E1 -12503.563,E2 -12503.563} C_VEL
LIN {X 0,Y 376.356,Z 384.602,A -85,B 0,C 180,E1 -12507.858,E2 -12507.858} C_VEL
LIN {X 0,Y 376.458,Z 384.59,A -85,B 0,C 180,E1 -12509.864,E2 -12509.864} C_VEL
LIN {X 0,Y 375.882,Z 384.668,A -85,B 0,C 180,E1 -12510.757,E2 -12510.757} C_VEL
LIN {X 0,Y 374.216,Z 384.88,A -85,B 0,C 180,E1 -12511.628,E2 -12511.628} C_VEL
LIN {X 0,Y 370.182,Z 385.381,A -85,B 0,C 180,E1 -12513.369,E2 -12513.369} C_VEL
LIN {X 0,Y 369.081,Z 385.513,A -85,B 0,C 180,E1 -12514.278,E2 -12514.278} C_VEL
LIN {X 0,Y 369.017,Z 385.518,A -85,B 0,C 180,E1 -12514.587,E2 -12514.587} C_VEL
LIN {X 0,Y 369.211,Z 385.494,A -85,B 0,C 180,E1 -12516.557,E2 -12516.557} C_VEL
LIN {X 0,Y 369.139,Z 385.501,A -85,B 0,C 180,E1 -12518.759,E2 -12518.759} C_VEL
LIN {X 0,Y 369.007,Z 385.523,A -85,B 0,C 180,E1 -12522.092,E2 -12522.092} C_VEL
LIN {X 0,Y 369.002,Z 385.518,A -85,B 0,C 180,E1 -12525.463,E2 -12525.463} C_VEL
LIN {X 0,Y 368.983,Z 385.519,A -85,B 0,C 180,E1 -12528.891,E2 -12528.891} C_VEL
LIN {X 0,Y 368.921,Z 385.529,A -85,B 0,C 180,E1 -12532.394,E2 -12532.394} C_VEL
LIN {X 0,Y 368.998,Z 385.522,A -85,B 0,C 180,E1 -12535.978,E2 -12535.978} C_VEL
LIN {X 0,Y 368.968,Z 385.521,A -85,B 0,C 180,E1 -12538.812,E2 -12538.812} C_VEL
LIN {X 0,Y 368.908,Z 385.53,A -85,B 0,C 180,E1 -12542.235,E2 -12542.235} C_VEL
LIN {X 0,Y 368.925,Z 385.527,A -85,B 0,C 180,E1 -12545,E2 -12545} C_VEL
LIN {X 0,Y 368.908,Z 385.529,A -85,B 0,C 180,E1 -12548.64,E2 -12548.64} C_VEL
LIN {X 0,Y 368.905,Z 385.532,A -85,B 0,C 180,E1 -12551.817,E2 -12551.817} C_VEL
LIN {X 0,Y 368.988,Z 385.646,A -85,B 0,C 180,E1 -12554.48,E2 -12554.48} C_VEL
LIN {X 0,Y 370.704,Z 394.723,A -85,B 0,C 180,E1 -12556.562,E2 -12556.562} C_VEL
LIN {X 0,Y 371.067,Z 397.5,A -85,B 0,C 180,E1 -12557.133,E2 -12557.133} C_VEL
LIN {X 0,Y 375.65,Z 423.334,A -85,B 0,C 180,E1 -12557.96,E2 -12557.96} C_VEL
LIN {X 0,Y 373.828,Z 506.743,A -85,B 0,C 180,E1 -12559.828,E2 -12559.828} C_VEL
LIN {X 0,Y 373.388,Z 518.639,A -85,B 0,C 180,E1 -12560.275,E2 -12560.275} C_VEL
LIN {X 0,Y 372.816,Z 531.077,A -85,B 0,C 180,E1 -12560.952,E2 -12560.952} C_VEL
LIN {X 0,Y 372.011,Z 544.017,A -85,B 0,C 180,E1 -12561.896,E2 -12561.896} C_VEL
LIN {X 0,Y 371.116,Z 555.969,A -85,B 0,C 180,E1 -12563.039,E2 -12563.039} C_VEL
LIN {X 0,Y 370.406,Z 565.677,A -85,B 0,C 180,E1 -12564.197,E2 -12564.197} C_VEL
LIN {X 0,Y 369.639,Z 575.014,A -85,B 0,C 180,E1 -12565.553,E2 -12565.553} C_VEL
LIN {X 0,Y 368.917,Z 583.754,A -85,B 0,C 180,E1 -12567.129,E2 -12567.129} C_VEL
LIN {X 0,Y 368.376,Z 590.704,A -85,B 0,C 180,E1 -12568.675,E2 -12568.675} C_VEL
LIN {X 0,Y 367.967,Z 596.343,A -85,B 0,C 180,E1 -12570.225,E2 -12570.225} C_VEL
LIN {X 0,Y 367.638,Z 601.677,A -85,B 0,C 180,E1 -12572.111,E2 -12572.111} C_VEL
LIN {X 0,Y 367.403,Z 605.565,A -85,B 0,C 180,E1 -12574.03,E2 -12574.03} C_VEL
LIN {X 0,Y 367.264,Z 607.15,A -85,B 0,C 180,E1 -12575.102,E2 -12575.102} C_VEL
LIN {X 0,Y 367.191,Z 608.738,A -85,B 0,C 180,E1 -12576.734,E2 -12576.734} C_VEL
LIN {X 0,Y 367.159,Z 609.429,A -85,B 0,C 180,E1 -12578.673,E2 -12578.673} C_VEL
LIN {X 0,Y 367.263,Z 609.174,A -85,B 0,C 180,E1 -12579.852,E2 -12579.852} C_VEL
LIN {X 0,Y 367.315,Z 608.484,A -85,B 0,C 180,E1 -12581.018,E2 -12581.018} C_VEL
LIN {X 0,Y 367.598,Z 606.303,A -85,B 0,C 180,E1 -12582.921,E2 -12582.921} C_VEL
LIN {X 0,Y 367.85,Z 603.524,A -85,B 0,C 180,E1 -12584.486,E2 -12584.486} C_VEL
LIN {X 0,Y 368.256,Z 599.368,A -85,B 0,C 180,E1 -12586.194,E2 -12586.194} C_VEL
LIN {X 0,Y 369.022,Z 592.872,A -85,B 0,C 180,E1 -12588.186,E2 -12588.186} C_VEL
LIN {X 0,Y 369.842,Z 585.782,A -85,B 0,C 180,E1 -12589.876,E2 -12589.876} C_VEL
LIN {X 0,Y 370.866,Z 576.921,A -85,B 0,C 180,E1 -12591.555,E2 -12591.555} C_VEL
LIN {X 0,Y 371.921,Z 567.819,A -85,B 0,C 180,E1 -12592.945,E2 -12592.945} C_VEL
LIN {X 0,Y 373.003,Z 557.73,A -85,B 0,C 180,E1 -12594.187,E2 -12594.187} C_VEL
LIN {X 0,Y 374.111,Z 546.455,A -85,B 0,C 180,E1 -12595.303,E2 -12595.303} C_VEL
LIN {X 0,Y 375.101,Z 534.332,A -85,B 0,C 180,E1 -12596.24,E2 -12596.24} C_VEL
LIN {X 0,Y 375.906,Z 521.481,A -85,B 0,C 180,E1 -12596.986,E2 -12596.986} C_VEL
LIN {X 0,Y 376.599,Z 508.842,A -85,B 0,C 180,E1 -12597.493,E2 -12597.493} C_VEL
LIN {X 0,Y 377.955,Z 462.933,A -85,B 0,C 180,E1 -12598.601,E2 -12598.601} C_VEL
LIN {X 0,Y 379.126,Z 424.494,A -85,B 0,C 180,E1 -12599.527,E2 -12599.527} C_VEL
LIN {X 0,Y 375.239,Z 406.319,A -85,B 0,C 180,E1 -12600.336,E2 -12600.336} C_VEL
LIN {X 0,Y 372.318,Z 398.477,A -85,B 0,C 180,E1 -12600.812,E2 -12600.812} C_VEL
LIN {X 0,Y 370.259,Z 389.571,A -85,B 0,C 180,E1 -12602.992,E2 -12602.992} C_VEL
LIN {X 0,Y 369.013,Z 385.524,A -85,B 0,C 180,E1 -12604.027,E2 -12604.027} C_VEL
LIN {X 0,Y 369.197,Z 385.498,A -85,B 0,C 180,E1 -12606.558,E2 -12606.558} C_VEL
LIN {X 0,Y 369.128,Z 385.506,A -85,B 0,C 180,E1 -12608.761,E2 -12608.761} C_VEL
LIN {X 0,Y 369.002,Z 385.52,A -85,B 0,C 180,E1 -12612.093,E2 -12612.093} C_VEL
LIN {X 0,Y 368.991,Z 385.523,A -85,B 0,C 180,E1 -12615.465,E2 -12615.465} C_VEL
LIN {X 0,Y 368.983,Z 385.523,A -85,B 0,C 180,E1 -12618.893,E2 -12618.893} C_VEL
LIN {X 0,Y 368.968,Z 385.524,A -85,B 0,C 180,E1 -12622.393,E2 -12622.393} C_VEL
LIN {X 0,Y 368.991,Z 385.522,A -85,B 0,C 180,E1 -12625.981,E2 -12625.981} C_VEL
LIN {X 0,Y 368.958,Z 385.525,A -85,B 0,C 180,E1 -12628.814,E2 -12628.814} C_VEL
LIN {X 0,Y 368.901,Z 385.533,A -85,B 0,C 180,E1 -12632.238,E2 -12632.238} C_VEL
LIN {X 0,Y 368.92,Z 385.531,A -85,B 0,C 180,E1 -12635.003,E2 -12635.003} C_VEL
LIN {X 0,Y 368.902,Z 385.532,A -85,B 0,C 180,E1 -12638.642,E2 -12638.642} C_VEL
LIN {X 0,Y 368.874,Z 385.535,A -85,B 0,C 180,E1 -12642.011,E2 -12642.011} C_VEL
LIN {X 0,Y 368.901,Z 385.535,A -85,B 0,C 180,E1 -12645.182,E2 -12645.182} C_VEL
LIN {X 0,Y 368.877,Z 385.535,A -85,B 0,C 180,E1 -12648.179,E2 -12648.179} C_VEL
LIN {X 0,Y 368.905,Z 385.534,A -85,B 0,C 180,E1 -12651.361,E2 -12651.361} C_VEL
LIN {X 0,Y 368.932,Z 385.53,A -85,B 0,C 180,E1 -12655.148,E2 -12655.148} C_VEL
LIN {X 0,Y 368.925,Z 385.531,A -85,B 0,C 180,E1 -12659.048,E2 -12659.048} C_VEL
LIN {X 0,Y 368.959,Z 385.53,A -85,B 0,C 180,E1 -12660.723,E2 -12660.723} C_VEL
LIN {X 0,Y 371.301,Z 396.692,A -85,B 0,C 180,E1 -12663.591,E2 -12663.591} C_VEL
LIN {X 0,Y 372.542,Z 404.333,A -85,B 0,C 180,E1 -12665.481,E2 -12665.481} C_VEL
LIN {X 0,Y 371.834,Z 412.569,A -85,B 0,C 180,E1 -12667.368,E2 -12667.368} C_VEL
LIN {X 0,Y 375.915,Z 434.567,A -85,B 0,C 180,E1 -12668.328,E2 -12668.328} C_VEL
LIN {X 0,Y 377.955,Z 451.409,A -85,B 0,C 180,E1 -12668.943,E2 -12668.943} C_VEL
LIN {X 0,Y 375.771,Z 527.393,A -85,B 0,C 180,E1 -12670.79,E2 -12670.79} C_VEL
LIN {X 0,Y 374.871,Z 541.395,A -85,B 0,C 180,E1 -12671.346,E2 -12671.346} C_VEL
LIN {X 0,Y 373.975,Z 553.845,A -85,B 0,C 180,E1 -12672.079,E2 -12672.079} C_VEL
LIN {X 0,Y 372.891,Z 565.938,A -85,B 0,C 180,E1 -12673.016,E2 -12673.016} C_VEL
LIN {X 0,Y 371.811,Z 576.843,A -85,B 0,C 180,E1 -12674.094,E2 -12674.094} C_VEL
LIN {X 0,Y 370.849,Z 586.75,A -85,B 0,C 180,E1 -12675.322,E2 -12675.322} C_VEL
LIN {X 0,Y 369.906,Z 596.575,A -85,B 0,C 180,E1 -12676.823,E2 -12676.823} C_VEL
LIN {X 0,Y 368.902,Z 605.174,A -85,B 0,C 180,E1 -12678.462,E2 -12678.462} C_VEL
LIN {X 0,Y 368.261,Z 612.083,A -85,B 0,C 180,E1 -12680.111,E2 -12680.111} C_VEL
LIN {X 0,Y 367.843,Z 617.786,A -85,B 0,C 180,E1 -12681.763,E2 -12681.763} C_VEL
LIN {X 0,Y 367.562,Z 622.39,A -85,B 0,C 180,E1 -12683.414,E2 -12683.414} C_VEL
LIN {X 0,Y 367.467,Z 624.802,A -85,B 0,C 180,E1 -12684.514,E2 -12684.514} C_VEL
LIN {X 0,Y 367.456,Z 626.776,A -85,B 0,C 180,E1 -12685.614,E2 -12685.614} C_VEL
LIN {X 0,Y 367.38,Z 628.324,A -85,B 0,C 180,E1 -12686.711,E2 -12686.711} C_VEL
LIN {X 0,Y 367.361,Z 629.412,A -85,B 0,C 180,E1 -12687.809,E2 -12687.809} C_VEL
LIN {X 0,Y 367.417,Z 630.092,A -85,B 0,C 180,E1 -12688.905,E2 -12688.905} C_VEL
LIN {X 0,Y 367.456,Z 630.377,A -85,B 0,C 180,E1 -12690.001,E2 -12690.001} C_VEL
LIN {X 0,Y 367.403,Z 630.265,A -85,B 0,C 180,E1 -12691.097,E2 -12691.097} C_VEL
LIN {X 0,Y 367.359,Z 629.712,A -85,B 0,C 180,E1 -12692.194,E2 -12692.194} C_VEL
LIN {X 0,Y 367.378,Z 628.754,A -85,B 0,C 180,E1 -12693.291,E2 -12693.291} C_VEL
LIN {X 0,Y 367.438,Z 627.398,A -85,B 0,C 180,E1 -12694.389,E2 -12694.389} C_VEL
LIN {X 0,Y 367.48,Z 624.58,A -85,B 0,C 180,E1 -12696.015,E2 -12696.015} C_VEL
LIN {X 0,Y 367.73,Z 620.633,A -85,B 0,C 180,E1 -12697.69,E2 -12697.69} C_VEL
LIN {X 0,Y 368.145,Z 615.605,A -85,B 0,C 180,E1 -12699.34,E2 -12699.34} C_VEL
LIN {X 0,Y 368.722,Z 609.295,A -85,B 0,C 180,E1 -12700.989,E2 -12700.989} C_VEL
LIN {X 0,Y 369.634,Z 601.421,A -85,B 0,C 180,E1 -12702.631,E2 -12702.631} C_VEL
LIN {X 0,Y 370.689,Z 591.599,A -85,B 0,C 180,E1 -12704.27,E2 -12704.27} C_VEL
LIN {X 0,Y 371.684,Z 581.437,A -85,B 0,C 180,E1 -12705.633,E2 -12705.633} C_VEL
LIN {X 0,Y 372.859,Z 569.956,A -85,B 0,C 180,E1 -12706.847,E2 -12706.847} C_VEL
LIN {X 0,Y 373.943,Z 558.716,A -85,B 0,C 180,E1 -12707.784,E2 -12707.784} C_VEL
LIN {X 0,Y 374.898,Z 546.113,A -85,B 0,C 180,E1 -12708.585,E2 -12708.585} C_VEL
LIN {X 0,Y 375.73,Z 532.758,A -85,B 0,C 180,E1 -12709.179,E2 -12709.179} C_VEL
LIN {X 0,Y 376.291,Z 519.765,A -85,B 0,C 180,E1 -12709.54,E2 -12709.54} C_VEL
LIN {X 0,Y 377.487,Z 449.963,A -85,B 0,C 180,E1 -12710.968,E2 -12710.968} C_VEL
LIN {X 0,Y 373.96,Z 427.981,A -85,B 0,C 180,E1 -12711.689,E2 -12711.689} C_VEL
LIN {X 0,Y 371.89,Z 417.413,A -85,B 0,C 180,E1 -12712.084,E2 -12712.084} C_VEL
LIN {X 0,Y 373.026,Z 406.021,A -85,B 0,C 180,E1 -12714.749,E2 -12714.749} C_VEL
LIN {X 0,Y 371.606,Z 397.373,A -85,B 0,C 180,E1 -12716.996,E2 -12716.996} C_VEL
LIN {X 0,Y 369.424,Z 387.742,A -85,B 0,C 180,E1 -12719.647,E2 -12719.647} C_VEL
LIN {X 0,Y 368.95,Z 385.529,A -85,B 0,C 180,E1 -12720.319,E2 -12720.319} C_VEL
LIN {X 0,Y 368.901,Z 385.535,A -85,B 0,C 180,E1 -12723.539,E2 -12723.539} C_VEL
LIN {X 0,Y 368.907,Z 385.535,A -85,B 0,C 180,E1 -12726.857,E2 -12726.857} C_VEL
LIN {X 0,Y 368.916,Z 385.534,A -85,B 0,C 180,E1 -12730.371,E2 -12730.371} C_VEL
LIN {X 0,Y 368.888,Z 385.537,A -85,B 0,C 180,E1 -12733.617,E2 -12733.617} C_VEL
LIN {X 0,Y 368.891,Z 385.535,A -85,B 0,C 180,E1 -12736.697,E2 -12736.697} C_VEL
LIN {X 0,Y 368.917,Z 385.525,A -85,B 0,C 180,E1 -12739.644,E2 -12739.644} C_VEL
LIN {X 0,Y 368.907,Z 385.53,A -85,B 0,C 180,E1 -12743.145,E2 -12743.145} C_VEL
LIN {X 0,Y 368.902,Z 385.528,A -85,B 0,C 180,E1 -12746.462,E2 -12746.462} C_VEL
LIN {X 0,Y 368.935,Z 385.522,A -85,B 0,C 180,E1 -12749.047,E2 -12749.047} C_VEL
LIN {X 0,Y 368.969,Z 385.519,A -85,B 0,C 180,E1 -12752.797,E2 -12752.797} C_VEL
LIN {X 0,Y 368.951,Z 385.527,A -85,B 0,C 180,E1 -12756.113,E2 -12756.113} C_VEL
LIN {X 0,Y 368.943,Z 385.528,A -85,B 0,C 180,E1 -12759.947,E2 -12759.947} C_VEL
LIN {X 0,Y 368.982,Z 385.521,A -85,B 0,C 180,E1 -12763.399,E2 -12763.399} C_VEL
LIN {X 0,Y 369.064,Z 385.513,A -85,B 0,C 180,E1 -12766.79,E2 -12766.79} C_VEL
LIN {X 0,Y 369.074,Z 385.506,A -85,B 0,C 180,E1 -12770.132,E2 -12770.132} C_VEL
LIN {X 0,Y 369.195,Z 385.494,A -85,B 0,C 180,E1 -12772.342,E2 -12772.342} C_VEL
LIN {X 0,Y 369.15,Z 385.503,A -85,B 0,C 180,E1 -12774.538,E2 -12774.538} C_VEL
LIN {X 0,Y 369.323,Z 385.475,A -85,B 0,C 180,E1 -12777.819,E2 -12777.819} C_VEL
LIN {X 0,Y 369.463,Z 385.461,A -85,B 0,C 180,E1 -12780,E2 -12780} C_VEL
LIN {X 0,Y 369.323,Z 385.483,A -85,B 0,C 180,E1 -12782.181,E2 -12782.181} C_VEL
LIN {X 0,Y 369.211,Z 385.49,A -85,B 0,C 180,E1 -12786.609,E2 -12786.609} C_VEL
LIN {X 0,Y 369.144,Z 385.502,A -85,B 0,C 180,E1 -12788.761,E2 -12788.761} C_VEL
LIN {X 0,Y 369.012,Z 385.519,A -85,B 0,C 180,E1 -12792.093,E2 -12792.093} C_VEL
LIN {X 0,Y 369.004,Z 385.523,A -85,B 0,C 180,E1 -12795.465,E2 -12795.465} C_VEL
LIN {X 0,Y 368.989,Z 385.524,A -85,B 0,C 180,E1 -12798.893,E2 -12798.893} C_VEL
LIN {X 0,Y 368.939,Z 385.53,A -85,B 0,C 180,E1 -12802.395,E2 -12802.395} C_VEL
LIN {X 0,Y 369.025,Z 385.614,A -85,B 0,C 180,E1 -12805.675,E2 -12805.675} C_VEL
LIN {X 0,Y 371.216,Z 395.985,A -85,B 0,C 180,E1 -12808.867,E2 -12808.867} C_VEL
LIN {X 0,Y 371.831,Z 399.835,A -85,B 0,C 180,E1 -12809.992,E2 -12809.992} C_VEL
LIN {X 0,Y 374.393,Z 407.698,A -85,B 0,C 180,E1 -12810.348,E2 -12810.348} C_VEL
LIN {X 0,Y 378.038,Z 424.983,A -85,B 0,C 180,E1 -12810.98,E2 -12810.98} C_VEL
LIN {X 0,Y 376.243,Z 507.199,A -85,B 0,C 180,E1 -12812.681,E2 -12812.681} C_VEL
LIN {X 0,Y 375.649,Z 520.582,A -85,B 0,C 180,E1 -12813.178,E2 -12813.178} C_VEL
LIN {X 0,Y 374.946,Z 532.262,A -85,B 0,C 180,E1 -12813.812,E2 -12813.812} C_VEL
LIN {X 0,Y 374.009,Z 544.656,A -85,B 0,C 180,E1 -12814.722,E2 -12814.722} C_VEL
LIN {X 0,Y 372.889,Z 556.568,A -85,B 0,C 180,E1 -12815.86,E2 -12815.86} C_VEL
LIN {X 0,Y 371.916,Z 566.392,A -85,B 0,C 180,E1 -12817.04,E2 -12817.04} C_VEL
LIN {X 0,Y 370.774,Z 576.055,A -85,B 0,C 180,E1 -12818.48,E2 -12818.48} C_VEL
LIN {X 0,Y 369.829,Z 584.322,A -85,B 0,C 180,E1 -12820.005,E2 -12820.005} C_VEL
LIN {X 0,Y 368.974,Z 592.14,A -85,B 0,C 180,E1 -12821.81,E2 -12821.81} C_VEL
LIN {X 0,Y 368.397,Z 597.961,A -85,B 0,C 180,E1 -12823.535,E2 -12823.535} C_VEL
LIN {X 0,Y 367.968,Z 601.975,A -85,B 0,C 180,E1 -12825.033,E2 -12825.033} C_VEL
LIN {X 0,Y 367.633,Z 605.195,A -85,B 0,C 180,E1 -12826.589,E2 -12826.589} C_VEL
LIN {X 0,Y 367.382,Z 607.636,A -85,B 0,C 180,E1 -12828.251,E2 -12828.251} C_VEL
LIN {X 0,Y 367.223,Z 609.144,A -85,B 0,C 180,E1 -12829.955,E2 -12829.955} C_VEL
LIN {X 0,Y 367.159,Z 609.681,A -85,B 0,C 180,E1 -12831.703,E2 -12831.703} C_VEL
LIN {X 0,Y 367.171,Z 609.116,A -85,B 0,C 180,E1 -12833.602,E2 -12833.602} C_VEL
LIN {X 0,Y 367.288,Z 607.496,A -85,B 0,C 180,E1 -12835.366,E2 -12835.366} C_VEL
LIN {X 0,Y 367.613,Z 604.515,A -85,B 0,C 180,E1 -12837.267,E2 -12837.267} C_VEL
LIN {X 0,Y 367.957,Z 599.945,A -85,B 0,C 180,E1 -12839.261,E2 -12839.261} C_VEL
LIN {X 0,Y 368.325,Z 595.2,A -85,B 0,C 180,E1 -12840.823,E2 -12840.823} C_VEL
LIN {X 0,Y 368.946,Z 588.864,A -85,B 0,C 180,E1 -12842.487,E2 -12842.487} C_VEL
LIN {X 0,Y 369.635,Z 581.359,A -85,B 0,C 180,E1 -12844.066,E2 -12844.066} C_VEL
LIN {X 0,Y 370.503,Z 572.453,A -85,B 0,C 180,E1 -12845.576,E2 -12845.576} C_VEL
LIN {X 0,Y 371.42,Z 562.986,A -85,B 0,C 180,E1 -12846.881,E2 -12846.881} C_VEL
LIN {X 0,Y 372.335,Z 551.93,A -85,B 0,C 180,E1 -12848.111,E2 -12848.111} C_VEL
LIN {X 0,Y 373.297,Z 539.749,A -85,B 0,C 180,E1 -12849.163,E2 -12849.163} C_VEL
LIN {X 0,Y 374.035,Z 527.653,A -85,B 0,C 180,E1 -12849.966,E2 -12849.966} C_VEL
LIN {X 0,Y 374.672,Z 514.486,A -85,B 0,C 180,E1 -12850.586,E2 -12850.586} C_VEL
LIN {X 0,Y 375.084,Z 500.561,A -85,B 0,C 180,E1 -12850.999,E2 -12850.999} C_VEL
LIN {X 0,Y 376.384,Z 423.202,A -85,B 0,C 180,E1 -12852.553,E2 -12852.553} C_VEL
LIN {X 0,Y 371.451,Z 398.879,A -85,B 0,C 180,E1 -12853.334,E2 -12853.334} C_VEL
LIN {X 0,Y 369.504,Z 387.733,A -85,B 0,C 180,E1 -12856.466,E2 -12856.466} C_VEL
LIN {X 0,Y 369.05,Z 385.516,A -85,B 0,C 180,E1 -12857.139,E2 -12857.139} C_VEL
LIN {X 0,Y 369.097,Z 385.505,A -85,B 0,C 180,E1 -12861.237,E2 -12861.237} C_VEL
LIN {X 0,Y 369.136,Z 385.506,A -85,B 0,C 180,E1 -12864.536,E2 -12864.536} C_VEL
LIN {X 0,Y 369.321,Z 385.478,A -85,B 0,C 180,E1 -12867.817,E2 -12867.817} C_VEL
LIN {X 0,Y 369.461,Z 385.463,A -85,B 0,C 180,E1 -12869.999,E2 -12869.999} C_VEL
LIN {X 0,Y 369.322,Z 385.482,A -85,B 0,C 180,E1 -12872.18,E2 -12872.18} C_VEL
LIN {X 0,Y 369.017,Z 385.518,A -85,B 0,C 180,E1 -12874.587,E2 -12874.587} C_VEL
LIN {X 0,Y 368.428,Z 385.59,A -85,B 0,C 180,E1 -12875.499,E2 -12875.499} C_VEL
LIN {X 0,Y 365.627,Z 385.938,A -85,B 0,C 180,E1 -12876.984,E2 -12876.984} C_VEL
LIN {X 0,Y 363.198,Z 386.246,A -85,B 0,C 180,E1 -12878.185,E2 -12878.185} C_VEL
LIN {X 0,Y 362.135,Z 386.373,A -85,B 0,C 180,E1 -12879.113,E2 -12879.113} C_VEL
LIN {X 0,Y 362.04,Z 386.385,A -85,B 0,C 180,E1 -12879.428,E2 -12879.428} C_VEL
LIN {X 0,Y 362,Z 386.39,A -85,B 0,C 180,E1 -12883.471,E2 -12883.471} C_VEL
LIN {X 0,Y 361.936,Z 386.397,A -85,B 0,C 180,E1 -12886.932,E2 -12886.932} C_VEL
LIN {X 0,Y 361.887,Z 386.405,A -85,B 0,C 180,E1 -12890.459,E2 -12890.459} C_VEL
LIN {X 0,Y 361.891,Z 386.407,A -85,B 0,C 180,E1 -12894.111,E2 -12894.111} C_VEL
LIN {X 0,Y 361.941,Z 386.397,A -85,B 0,C 180,E1 -12896.72,E2 -12896.72} C_VEL
LIN {X 0,Y 361.876,Z 386.406,A -85,B 0,C 180,E1 -12900.326,E2 -12900.326} C_VEL
LIN {X 0,Y 361.852,Z 386.409,A -85,B 0,C 180,E1 -12904.278,E2 -12904.278} C_VEL
LIN {X 0,Y 361.868,Z 386.408,A -85,B 0,C 180,E1 -12907.223,E2 -12907.223} C_VEL
LIN {X 0,Y 361.867,Z 386.406,A -85,B 0,C 180,E1 -12910.761,E2 -12910.761} C_VEL
LIN {X 0,Y 361.92,Z 386.408,A -85,B 0,C 180,E1 -12914.255,E2 -12914.255} C_VEL
LIN {X 0,Y 363.943,Z 397.389,A -85,B 0,C 180,E1 -12916.798,E2 -12916.798} C_VEL
LIN {X 0,Y 368.825,Z 424.163,A -85,B 0,C 180,E1 -12917.674,E2 -12917.674} C_VEL
LIN {X 0,Y 366.929,Z 506.496,A -85,B 0,C 180,E1 -12919.565,E2 -12919.565} C_VEL
LIN {X 0,Y 366.48,Z 518.215,A -85,B 0,C 180,E1 -12920.008,E2 -12920.008} C_VEL
LIN {X 0,Y 365.924,Z 530.389,A -85,B 0,C 180,E1 -12920.668,E2 -12920.668} C_VEL
LIN {X 0,Y 365.089,Z 543.425,A -85,B 0,C 180,E1 -12921.624,E2 -12921.624} C_VEL
LIN {X 0,Y 364.221,Z 555.143,A -85,B 0,C 180,E1 -12922.741,E2 -12922.741} C_VEL
LIN {X 0,Y 363.385,Z 565.876,A -85,B 0,C 180,E1 -12924.033,E2 -12924.033} C_VEL
LIN {X 0,Y 362.588,Z 575.495,A -85,B 0,C 180,E1 -12925.462,E2 -12925.462} C_VEL
LIN {X 0,Y 361.862,Z 584.126,A -85,B 0,C 180,E1 -12927.056,E2 -12927.056} C_VEL
LIN {X 0,Y 361.286,Z 591.11,A -85,B 0,C 180,E1 -12928.646,E2 -12928.646} C_VEL
LIN {X 0,Y 360.878,Z 596.71,A -85,B 0,C 180,E1 -12930.224,E2 -12930.224} C_VEL
LIN {X 0,Y 360.556,Z 601.906,A -85,B 0,C 180,E1 -12932.107,E2 -12932.107} C_VEL
LIN {X 0,Y 360.354,Z 605.323,A -85,B 0,C 180,E1 -12933.78,E2 -12933.78} C_VEL
LIN {X 0,Y 360.103,Z 608.087,A -85,B 0,C 180,E1 -12935.804,E2 -12935.804} C_VEL
LIN {X 0,Y 360.083,Z 609.092,A -85,B 0,C 180,E1 -12937.023,E2 -12937.023} C_VEL
LIN {X 0,Y 360.065,Z 609.548,A -85,B 0,C 180,E1 -12938.231,E2 -12938.231} C_VEL
LIN {X 0,Y 360.13,Z 609.541,A -85,B 0,C 180,E1 -12939.504,E2 -12939.504} C_VEL
LIN {X 0,Y 360.209,Z 609.05,A -85,B 0,C 180,E1 -12940.629,E2 -12940.629} C_VEL
LIN {X 0,Y 360.484,Z 606.911,A -85,B 0,C 180,E1 -12942.798,E2 -12942.798} C_VEL
LIN {X 0,Y 360.834,Z 603.581,A -85,B 0,C 180,E1 -12944.755,E2 -12944.755} C_VEL
LIN {X 0,Y 361.307,Z 599.254,A -85,B 0,C 180,E1 -12946.543,E2 -12946.543} C_VEL
LIN {X 0,Y 362.106,Z 592.875,A -85,B 0,C 180,E1 -12948.525,E2 -12948.525} C_VEL
LIN {X 0,Y 362.977,Z 585.909,A -85,B 0,C 180,E1 -12950.207,E2 -12950.207} C_VEL
LIN {X 0,Y 364.141,Z 576.77,A -85,B 0,C 180,E1 -12951.956,E2 -12951.956} C_VEL
LIN {X 0,Y 365.256,Z 567.56,A -85,B 0,C 180,E1 -12953.37,E2 -12953.37} C_VEL
LIN {X 0,Y 366.253,Z 558.622,A -85,B 0,C 180,E1 -12954.494,E2 -12954.494} C_VEL
LIN {X 0,Y 367.556,Z 546.183,A -85,B 0,C 180,E1 -12955.751,E2 -12955.751} C_VEL
LIN {X 0,Y 368.604,Z 533.704,A -85,B 0,C 180,E1 -12956.721,E2 -12956.721} C_VEL
LIN {X 0,Y 369.493,Z 520.662,A -85,B 0,C 180,E1 -12957.479,E2 -12957.479} C_VEL
LIN {X 0,Y 370.204,Z 507.502,A -85,B 0,C 180,E1 -12957.994,E2 -12957.994} C_VEL
LIN {X 0,Y 372.817,Z 425.754,A -85,B 0,C 180,E1 -12960,E2 -12960} C_VEL
LIN {X 0,Y 369.399,Z 409.372,A -85,B 0,C 180,E1 -12960.761,E2 -12960.761} C_VEL
LIN {X 0,Y 366.601,Z 401.824,A -85,B 0,C 180,E1 -12961.233,E2 -12961.233} C_VEL
LIN {X 0,Y 365.179,Z 398.552,A -85,B 0,C 180,E1 -12961.482,E2 -12961.482} C_VEL
LIN {X 0,Y 363.078,Z 390.2,A -85,B 0,C 180,E1 -12963.607,E2 -12963.607} C_VEL
LIN {X 0,Y 361.988,Z 386.4,A -85,B 0,C 180,E1 -12964.593,E2 -12964.593} C_VEL
LIN {X 0,Y 362.161,Z 386.374,A -85,B 0,C 180,E1 -12966.686,E2 -12966.686} C_VEL
LIN {X 0,Y 362.065,Z 386.387,A -85,B 0,C 180,E1 -12968.933,E2 -12968.933} C_VEL
LIN {X 0,Y 361.956,Z 386.397,A -85,B 0,C 180,E1 -12972.332,E2 -12972.332} C_VEL
LIN {X 0,Y 361.953,Z 386.401,A -85,B 0,C 180,E1 -12974.621,E2 -12974.621} C_VEL
LIN {X 0,Y 361.951,Z 386.4,A -85,B 0,C 180,E1 -12978.1,E2 -12978.1} C_VEL
LIN {X 0,Y 361.922,Z 386.403,A -85,B 0,C 180,E1 -12981.651,E2 -12981.651} C_VEL
LIN {X 0,Y 361.921,Z 386.402,A -85,B 0,C 180,E1 -12985.291,E2 -12985.291} C_VEL
LIN {X 0,Y 361.913,Z 386.404,A -85,B 0,C 180,E1 -12987.779,E2 -12987.779} C_VEL
LIN {X 0,Y 361.851,Z 386.411,A -85,B 0,C 180,E1 -12991.628,E2 -12991.628} C_VEL
LIN {X 0,Y 361.866,Z 386.409,A -85,B 0,C 180,E1 -12995.346,E2 -12995.346} C_VEL
LIN {X 0,Y 361.863,Z 386.409,A -85,B 0,C 180,E1 -12999.028,E2 -12999.028} C_VEL
LIN {X 0,Y 361.83,Z 386.413,A -85,B 0,C 180,E1 -13002.83,E2 -13002.83} C_VEL
LIN {X 0,Y 361.823,Z 386.413,A -85,B 0,C 180,E1 -13005.946,E2 -13005.946} C_VEL
LIN {X 0,Y 361.83,Z 386.414,A -85,B 0,C 180,E1 -13009.246,E2 -13009.246} C_VEL
LIN {X 0,Y 361.86,Z 386.41,A -85,B 0,C 180,E1 -13012.778,E2 -13012.778} C_VEL
LIN {X 0,Y 361.851,Z 386.412,A -85,B 0,C 180,E1 -13015.721,E2 -13015.721} C_VEL
LIN {X 0,Y 361.88,Z 386.409,A -85,B 0,C 180,E1 -13019.675,E2 -13019.675} C_VEL
LIN {X 0,Y 361.947,Z 386.547,A -85,B 0,C 180,E1 -13020.456,E2 -13020.456} C_VEL
LIN {X 0,Y 364.121,Z 396.971,A -85,B 0,C 180,E1 -13023.196,E2 -13023.196} C_VEL
LIN {X 0,Y 365.561,Z 405.232,A -85,B 0,C 180,E1 -13025.284,E2 -13025.284} C_VEL
LIN {X 0,Y 365.067,Z 411.374,A -85,B 0,C 180,E1 -13026.724,E2 -13026.724} C_VEL
LIN {X 0,Y 369.696,Z 435.877,A -85,B 0,C 180,E1 -13027.849,E2 -13027.849} C_VEL
LIN {X 0,Y 371.621,Z 452.181,A -85,B 0,C 180,E1 -13028.467,E2 -13028.467} C_VEL
LIN {X 0,Y 369.272,Z 527.894,A -85,B 0,C 180,E1 -13030.366,E2 -13030.366} C_VEL
LIN {X 0,Y 368.313,Z 541.642,A -85,B 0,C 180,E1 -13030.929,E2 -13030.929} C_VEL
LIN {X 0,Y 367.285,Z 554.912,A -85,B 0,C 180,E1 -13031.741,E2 -13031.741} C_VEL
LIN {X 0,Y 366.153,Z 566.707,A -85,B 0,C 180,E1 -13032.694,E2 -13032.694} C_VEL
LIN {X 0,Y 364.906,Z 578.504,A -85,B 0,C 180,E1 -13033.929,E2 -13033.929} C_VEL
LIN {X 0,Y 363.843,Z 588.818,A -85,B 0,C 180,E1 -13035.284,E2 -13035.284} C_VEL
LIN {X 0,Y 362.796,Z 598.352,A -85,B 0,C 180,E1 -13036.845,E2 -13036.845} C_VEL
LIN {X 0,Y 361.785,Z 606.599,A -85,B 0,C 180,E1 -13038.516,E2 -13038.516} C_VEL
LIN {X 0,Y 361.24,Z 612.187,A -85,B 0,C 180,E1 -13039.917,E2 -13039.917} C_VEL
LIN {X 0,Y 360.791,Z 617.641,A -85,B 0,C 180,E1 -13041.601,E2 -13041.601} C_VEL
LIN {X 0,Y 360.431,Z 623.623,A -85,B 0,C 180,E1 -13043.958,E2 -13043.958} C_VEL
LIN {X 0,Y 360.365,Z 626.52,A -85,B 0,C 180,E1 -13045.527,E2 -13045.527} C_VEL
LIN {X 0,Y 360.3,Z 628.081,A -85,B 0,C 180,E1 -13046.647,E2 -13046.647} C_VEL
LIN {X 0,Y 360.265,Z 629.187,A -85,B 0,C 180,E1 -13047.765,E2 -13047.765} C_VEL
LIN {X 0,Y 360.317,Z 629.876,A -85,B 0,C 180,E1 -13048.884,E2 -13048.884} C_VEL
LIN {X 0,Y 360.359,Z 630.171,A -85,B 0,C 180,E1 -13050.001,E2 -13050.001} C_VEL
LIN {X 0,Y 360.303,Z 630.069,A -85,B 0,C 180,E1 -13051.119,E2 -13051.119} C_VEL
LIN {X 0,Y 360.263,Z 629.533,A -85,B 0,C 180,E1 -13052.237,E2 -13052.237} C_VEL
LIN {X 0,Y 360.297,Z 628.586,A -85,B 0,C 180,E1 -13053.356,E2 -13053.356} C_VEL
LIN {X 0,Y 360.349,Z 627.24,A -85,B 0,C 180,E1 -13054.476,E2 -13054.476} C_VEL
LIN {X 0,Y 360.379,Z 624.778,A -85,B 0,C 180,E1 -13055.963,E2 -13055.963} C_VEL
LIN {X 0,Y 360.681,Z 620.524,A -85,B 0,C 180,E1 -13057.841,E2 -13057.841} C_VEL
LIN {X 0,Y 361.099,Z 615.518,A -85,B 0,C 180,E1 -13059.524,E2 -13059.524} C_VEL
LIN {X 0,Y 361.71,Z 609.232,A -85,B 0,C 180,E1 -13061.205,E2 -13061.205} C_VEL
LIN {X 0,Y 362.691,Z 601.401,A -85,B 0,C 180,E1 -13062.877,E2 -13062.877} C_VEL
LIN {X 0,Y 363.634,Z 593.409,A -85,B 0,C 180,E1 -13064.267,E2 -13064.267} C_VEL
LIN {X 0,Y 364.629,Z 583.675,A -85,B 0,C 180,E1 -13065.656,E2 -13065.656} C_VEL
LIN {X 0,Y 365.789,Z 572.892,A -85,B 0,C 180,E1 -13066.895,E2 -13066.895} C_VEL
LIN {X 0,Y 366.889,Z 562.45,A -85,B 0,C 180,E1 -13067.849,E2 -13067.849} C_VEL
LIN {X 0,Y 367.953,Z 549.982,A -85,B 0,C 180,E1 -13068.732,E2 -13068.732} C_VEL
LIN {X 0,Y 368.85,Z 536.951,A -85,B 0,C 180,E1 -13069.407,E2 -13069.407} C_VEL
LIN {X 0,Y 369.596,Z 524.083,A -85,B 0,C 180,E1 -13069.836,E2 -13069.836} C_VEL
LIN {X 0,Y 370.967,Z 450.973,A -85,B 0,C 180,E1 -13071.379,E2 -13071.379} C_VEL
LIN {X 0,Y 367.498,Z 429.08,A -85,B 0,C 180,E1 -13072.113,E2 -13072.113} C_VEL
LIN {X 0,Y 365.121,Z 417.245,A -85,B 0,C 180,E1 -13072.564,E2 -13072.564} C_VEL
LIN {X 0,Y 366.133,Z 407.15,A -85,B 0,C 180,E1 -13074.981,E2 -13074.981} C_VEL
LIN {X 0,Y 364.42,Z 397.466,A -85,B 0,C 180,E1 -13077.573,E2 -13077.573} C_VEL
LIN {X 0,Y 361.89,Z 386.409,A -85,B 0,C 180,E1 -13080.748,E2 -13080.748} C_VEL
LIN {X 0,Y 361.859,Z 386.41,A -85,B 0,C 180,E1 -13084.281,E2 -13084.281} C_VEL
LIN {X 0,Y 361.869,Z 386.413,A -85,B 0,C 180,E1 -13087.224,E2 -13087.224} C_VEL
LIN {X 0,Y 361.841,Z 386.416,A -85,B 0,C 180,E1 -13090.756,E2 -13090.756} C_VEL
LIN {X 0,Y 361.823,Z 386.417,A -85,B 0,C 180,E1 -13094.369,E2 -13094.369} C_VEL
LIN {X 0,Y 361.842,Z 386.412,A -85,B 0,C 180,E1 -13097.569,E2 -13097.569} C_VEL
LIN {X 0,Y 361.875,Z 386.41,A -85,B 0,C 180,E1 -13100.974,E2 -13100.974} C_VEL
LIN {X 0,Y 361.88,Z 386.41,A -85,B 0,C 180,E1 -13104.656,E2 -13104.656} C_VEL
LIN {X 0,Y 361.844,Z 386.413,A -85,B 0,C 180,E1 -13108.371,E2 -13108.371} C_VEL
LIN {X 0,Y 361.914,Z 386.403,A -85,B 0,C 180,E1 -13112.221,E2 -13112.221} C_VEL
LIN {X 0,Y 361.934,Z 386.401,A -85,B 0,C 180,E1 -13114.71,E2 -13114.71} C_VEL
LIN {X 0,Y 361.9,Z 386.401,A -85,B 0,C 180,E1 -13118.348,E2 -13118.348} C_VEL
LIN {X 0,Y 361.974,Z 386.389,A -85,B 0,C 180,E1 -13122.062,E2 -13122.062} C_VEL
LIN {X 0,Y 362.004,Z 386.385,A -85,B 0,C 180,E1 -13126.102,E2 -13126.102} C_VEL
LIN {X 0,Y 362.038,Z 386.381,A -85,B 0,C 180,E1 -13129.938,E2 -13129.938} C_VEL
LIN {X 0,Y 362.158,Z 386.372,A -85,B 0,C 180,E1 -13132.193,E2 -13132.193} C_VEL
LIN {X 0,Y 362.124,Z 386.376,A -85,B 0,C 180,E1 -13134.431,E2 -13134.431} C_VEL
LIN {X 0,Y 362.287,Z 386.351,A -85,B 0,C 180,E1 -13137.777,E2 -13137.777} C_VEL
LIN {X 0,Y 362.433,Z 386.336,A -85,B 0,C 180,E1 -13140,E2 -13140} C_VEL
LIN {X 0,Y 362.287,Z 386.359,A -85,B 0,C 180,E1 -13142.224,E2 -13142.224} C_VEL
LIN {X 0,Y 362.179,Z 386.366,A -85,B 0,C 180,E1 -13146.686,E2 -13146.686} C_VEL
LIN {X 0,Y 362.081,Z 386.382,A -85,B 0,C 180,E1 -13148.933,E2 -13148.933} C_VEL
LIN {X 0,Y 361.967,Z 386.397,A -85,B 0,C 180,E1 -13152.332,E2 -13152.332} C_VEL
LIN {X 0,Y 361.969,Z 386.396,A -85,B 0,C 180,E1 -13154.62,E2 -13154.62} C_VEL
LIN {X 0,Y 361.967,Z 386.399,A -85,B 0,C 180,E1 -13158.099,E2 -13158.099} C_VEL
LIN {X 0,Y 361.899,Z 386.408,A -85,B 0,C 180,E1 -13161.653,E2 -13161.653} C_VEL
LIN {X 0,Y 361.946,Z 386.428,A -85,B 0,C 180,E1 -13165.212,E2 -13165.212} C_VEL
LIN {X 0,Y 363.998,Z 395.967,A -85,B 0,C 180,E1 -13168.232,E2 -13168.232} C_VEL
LIN {X 0,Y 364.771,Z 400.009,A -85,B 0,C 180,E1 -13169.467,E2 -13169.467} C_VEL
LIN {X 0,Y 367.861,Z 408.785,A -85,B 0,C 180,E1 -13169.911,E2 -13169.911} C_VEL
LIN {X 0,Y 371.517,Z 425.913,A -85,B 0,C 180,E1 -13170.557,E2 -13170.557} C_VEL
LIN {X 0,Y 369.67,Z 507.141,A -85,B 0,C 180,E1 -13172.27,E2 -13172.27} C_VEL
LIN {X 0,Y 369.058,Z 520.618,A -85,B 0,C 180,E1 -13172.778,E2 -13172.778} C_VEL
LIN {X 0,Y 368.218,Z 533.826,A -85,B 0,C 180,E1 -13173.52,E2 -13173.52} C_VEL
LIN {X 0,Y 367.197,Z 546.239,A -85,B 0,C 180,E1 -13174.479,E2 -13174.479} C_VEL
LIN {X 0,Y 366.146,Z 556.58,A -85,B 0,C 180,E1 -13175.495,E2 -13175.495} C_VEL
LIN {X 0,Y 365.018,Z 567.319,A -85,B 0,C 180,E1 -13176.818,E2 -13176.818} C_VEL
LIN {X 0,Y 363.915,Z 576.186,A -85,B 0,C 180,E1 -13178.17,E2 -13178.17} C_VEL
LIN {X 0,Y 362.927,Z 584.454,A -85,B 0,C 180,E1 -13179.72,E2 -13179.72} C_VEL
LIN {X 0,Y 362.04,Z 592.302,A -85,B 0,C 180,E1 -13181.563,E2 -13181.563} C_VEL
LIN {X 0,Y 361.373,Z 598.397,A -85,B 0,C 180,E1 -13183.412,E2 -13183.412} C_VEL
LIN {X 0,Y 360.792,Z 603.534,A -85,B 0,C 180,E1 -13185.471,E2 -13185.471} C_VEL
LIN {X 0,Y 360.475,Z 606.239,A -85,B 0,C 180,E1 -13186.969,E2 -13186.969} C_VEL
LIN {X 0,Y 360.259,Z 608.165,A -85,B 0,C 180,E1 -13188.448,E2 -13188.448} C_VEL
LIN {X 0,Y 360.156,Z 609.371,A -85,B 0,C 180,E1 -13189.911,E2 -13189.911} C_VEL
LIN {X 0,Y 360.084,Z 609.845,A -85,B 0,C 180,E1 -13191.348,E2 -13191.348} C_VEL
LIN {X 0,Y 360.054,Z 609.528,A -85,B 0,C 180,E1 -13193.158,E2 -13193.158} C_VEL
LIN {X 0,Y 360.162,Z 608.078,A -85,B 0,C 180,E1 -13195.042,E2 -13195.042} C_VEL
LIN {X 0,Y 360.476,Z 605.386,A -85,B 0,C 180,E1 -13196.967,E2 -13196.967} C_VEL
LIN {X 0,Y 360.835,Z 601.129,A -85,B 0,C 180,E1 -13198.981,E2 -13198.981} C_VEL
LIN {X 0,Y 361.268,Z 595.585,A -85,B 0,C 180,E1 -13200.898,E2 -13200.898} C_VEL
LIN {X 0,Y 361.974,Z 588.615,A -85,B 0,C 180,E1 -13202.757,E2 -13202.757} C_VEL
LIN {X 0,Y 362.75,Z 580.458,A -85,B 0,C 180,E1 -13204.463,E2 -13204.463} C_VEL
LIN {X 0,Y 363.704,Z 570.955,A -85,B 0,C 180,E1 -13206.058,E2 -13206.058} C_VEL
LIN {X 0,Y 364.68,Z 561.557,A -85,B 0,C 180,E1 -13207.328,E2 -13207.328} C_VEL
LIN {X 0,Y 365.607,Z 550.042,A -85,B 0,C 180,E1 -13208.577,E2 -13208.577} C_VEL
LIN {X 0,Y 366.599,Z 538.047,A -85,B 0,C 180,E1 -13209.593,E2 -13209.593} C_VEL
LIN {X 0,Y 367.307,Z 526.041,A -85,B 0,C 180,E1 -13210.363,E2 -13210.363} C_VEL
LIN {X 0,Y 367.965,Z 512.439,A -85,B 0,C 180,E1 -13210.979,E2 -13210.979} C_VEL
LIN {X 0,Y 368.353,Z 498.561,A -85,B 0,C 180,E1 -13211.361,E2 -13211.361} C_VEL
LIN {X 0,Y 369.691,Z 424.355,A -85,B 0,C 180,E1 -13212.879,E2 -13212.879} C_VEL
LIN {X 0,Y 365.061,Z 401.423,A -85,B 0,C 180,E1 -13213.632,E2 -13213.632} C_VEL
LIN {X 0,Y 364.306,Z 398.962,A -85,B 0,C 180,E1 -13213.755,E2 -13213.755} C_VEL
LIN {X 0,Y 362.569,Z 389.227,A -85,B 0,C 180,E1 -13216.548,E2 -13216.548} C_VEL
LIN {X 0,Y 362.015,Z 386.391,A -85,B 0,C 180,E1 -13217.383,E2 -13217.383} C_VEL
LIN {X 0,Y 362.052,Z 386.384,A -85,B 0,C 180,E1 -13221.065,E2 -13221.065} C_VEL
LIN {X 0,Y 362.108,Z 386.382,A -85,B 0,C 180,E1 -13224.43,E2 -13224.43} C_VEL
LIN {X 0,Y 362.285,Z 386.355,A -85,B 0,C 180,E1 -13227.775,E2 -13227.775} C_VEL
LIN {X 0,Y 362.43,Z 386.339,A -85,B 0,C 180,E1 -13229.999,E2 -13229.999} C_VEL
LIN {X 0,Y 362.286,Z 386.359,A -85,B 0,C 180,E1 -13232.222,E2 -13232.222} C_VEL
LIN {X 0,Y 362.175,Z 386.369,A -85,B 0,C 180,E1 -13236.685,E2 -13236.685} C_VEL
LIN {X 0,Y 362.04,Z 386.385,A -85,B 0,C 180,E1 -13239.428,E2 -13239.428} C_VEL
LIN {X 0,Y 361.35,Z 386.476,A -85,B 0,C 180,E1 -13240.356,E2 -13240.356} C_VEL
LIN {X 0,Y 358.486,Z 386.837,A -85,B 0,C 180,E1 -13241.866,E2 -13241.866} C_VEL
LIN {X 0,Y 356.066,Z 387.138,A -85,B 0,C 180,E1 -13243.088,E2 -13243.088} C_VEL
LIN {X 0,Y 355.017,Z 387.265,A -85,B 0,C 180,E1 -13244.032,E2 -13244.032} C_VEL
LIN {X 0,Y 354.926,Z 387.273,A -85,B 0,C 180,E1 -13244.353,E2 -13244.353} C_VEL
LIN {X 0,Y 354.906,Z 387.275,A -85,B 0,C 180,E1 -13248.47,E2 -13248.47} C_VEL
LIN {X 0,Y 354.824,Z 387.287,A -85,B 0,C 180,E1 -13252.105,E2 -13252.105} C_VEL
LIN {X 0,Y 354.897,Z 387.28,A -85,B 0,C 180,E1 -13255.826,E2 -13255.826} C_VEL
LIN {X 0,Y 354.852,Z 387.285,A -85,B 0,C 180,E1 -13259.677,E2 -13259.677} C_VEL
LIN {X 0,Y 354.827,Z 387.289,A -85,B 0,C 180,E1 -13263.68,E2 -13263.68} C_VEL
LIN {X 0,Y 354.797,Z 387.287,A -85,B 0,C 180,E1 -13266.457,E2 -13266.457} C_VEL
LIN {X 0,Y 354.819,Z 387.288,A -85,B 0,C 180,E1 -13269.422,E2 -13269.422} C_VEL
LIN {X 0,Y 354.805,Z 387.286,A -85,B 0,C 180,E1 -13272.87,E2 -13272.87} C_VEL
LIN {X 0,Y 354.865,Z 387.424,A -85,B 0,C 180,E1 -13274.074,E2 -13274.074} C_VEL
LIN {X 0,Y 356.802,Z 397.516,A -85,B 0,C 180,E1 -13276.451,E2 -13276.451} C_VEL
LIN {X 0,Y 358.703,Z 406.309,A -85,B 0,C 180,E1 -13276.767,E2 -13276.767} C_VEL
LIN {X 0,Y 361.993,Z 424.941,A -85,B 0,C 180,E1 -13277.384,E2 -13277.384} C_VEL
LIN {X 0,Y 359.991,Z 507.271,A -85,B 0,C 180,E1 -13279.325,E2 -13279.325} C_VEL
LIN {X 0,Y 359.546,Z 519.875,A -85,B 0,C 180,E1 -13279.831,E2 -13279.831} C_VEL
LIN {X 0,Y 358.771,Z 533.665,A -85,B 0,C 180,E1 -13280.639,E2 -13280.639} C_VEL
LIN {X 0,Y 357.977,Z 545.822,A -85,B 0,C 180,E1 -13281.601,E2 -13281.601} C_VEL
LIN {X 0,Y 357.119,Z 557.23,A -85,B 0,C 180,E1 -13282.76,E2 -13282.76} C_VEL
LIN {X 0,Y 356.306,Z 566.85,A -85,B 0,C 180,E1 -13283.967,E2 -13283.967} C_VEL
LIN {X 0,Y 355.521,Z 575.922,A -85,B 0,C 180,E1 -13285.359,E2 -13285.359} C_VEL
LIN {X 0,Y 354.782,Z 584.557,A -85,B 0,C 180,E1 -13286.992,E2 -13286.992} C_VEL
LIN {X 0,Y 354.239,Z 591.248,A -85,B 0,C 180,E1 -13288.548,E2 -13288.548} C_VEL
LIN {X 0,Y 353.782,Z 597.077,A -85,B 0,C 180,E1 -13290.222,E2 -13290.222} C_VEL
LIN {X 0,Y 353.47,Z 602.224,A -85,B 0,C 180,E1 -13292.144,E2 -13292.144} C_VEL
LIN {X 0,Y 353.204,Z 605.919,A -85,B 0,C 180,E1 -13294.039,E2 -13294.039} C_VEL
LIN {X 0,Y 353.058,Z 607.692,A -85,B 0,C 180,E1 -13295.29,E2 -13295.29} C_VEL
LIN {X 0,Y 353.008,Z 608.885,A -85,B 0,C 180,E1 -13296.535,E2 -13296.535} C_VEL
LIN {X 0,Y 352.957,Z 609.603,A -85,B 0,C 180,E1 -13297.77,E2 -13297.77} C_VEL
LIN {X 0,Y 353.015,Z 609.771,A -85,B 0,C 180,E1 -13299.336,E2 -13299.336} C_VEL
LIN {X 0,Y 353.192,Z 608.792,A -85,B 0,C 180,E1 -13301.435,E2 -13301.435} C_VEL
LIN {X 0,Y 353.374,Z 607.51,A -85,B 0,C 180,E1 -13302.67,E2 -13302.67} C_VEL
LIN {X 0,Y 353.686,Z 604.817,A -85,B 0,C 180,E1 -13304.439,E2 -13304.439} C_VEL
LIN {X 0,Y 354.208,Z 600.396,A -85,B 0,C 180,E1 -13306.458,E2 -13306.458} C_VEL
LIN {X 0,Y 354.827,Z 595.908,A -85,B 0,C 180,E1 -13307.996,E2 -13307.996} C_VEL
LIN {X 0,Y 355.654,Z 589.487,A -85,B 0,C 180,E1 -13309.755,E2 -13309.755} C_VEL
LIN {X 0,Y 356.75,Z 581.389,A -85,B 0,C 180,E1 -13311.503,E2 -13311.503} C_VEL
LIN {X 0,Y 357.836,Z 573.167,A -85,B 0,C 180,E1 -13312.949,E2 -13312.949} C_VEL
LIN {X 0,Y 359.077,Z 563.12,A -85,B 0,C 180,E1 -13314.384,E2 -13314.384} C_VEL
LIN {X 0,Y 360.413,Z 551.827,A -85,B 0,C 180,E1 -13315.666,E2 -13315.666} C_VEL
LIN {X 0,Y 361.518,Z 540.884,A -85,B 0,C 180,E1 -13316.656,E2 -13316.656} C_VEL
LIN {X 0,Y 362.6,Z 527.649,A -85,B 0,C 180,E1 -13317.57,E2 -13317.57} C_VEL
LIN {X 0,Y 363.376,Z 515.195,A -85,B 0,C 180,E1 -13318.199,E2 -13318.199} C_VEL
LIN {X 0,Y 364.023,Z 501.173,A -85,B 0,C 180,E1 -13318.652,E2 -13318.652} C_VEL
LIN {X 0,Y 366.534,Z 426.614,A -85,B 0,C 180,E1 -13320.521,E2 -13320.521} C_VEL
LIN {X 0,Y 363.25,Z 411.012,A -85,B 0,C 180,E1 -13321.276,E2 -13321.276} C_VEL
LIN {X 0,Y 359.494,Z 401.944,A -85,B 0,C 180,E1 -13321.912,E2 -13321.912} C_VEL
LIN {X 0,Y 358.104,Z 398.765,A -85,B 0,C 180,E1 -13322.179,E2 -13322.179} C_VEL
LIN {X 0,Y 356.202,Z 391.976,A -85,B 0,C 180,E1 -13323.96,E2 -13323.96} C_VEL
LIN {X 0,Y 355.004,Z 387.267,A -85,B 0,C 180,E1 -13325.253,E2 -13325.253} C_VEL
LIN {X 0,Y 355.117,Z 387.249,A -85,B 0,C 180,E1 -13328.311,E2 -13328.311} C_VEL
LIN {X 0,Y 354.915,Z 387.274,A -85,B 0,C 180,E1 -13332.581,E2 -13332.581} C_VEL
LIN {X 0,Y 354.882,Z 387.283,A -85,B 0,C 180,E1 -13336.096,E2 -13336.096} C_VEL
LIN {X 0,Y 354.9,Z 387.279,A -85,B 0,C 180,E1 -13338.472,E2 -13338.472} C_VEL
LIN {X 0,Y 354.882,Z 387.281,A -85,B 0,C 180,E1 -13342.103,E2 -13342.103} C_VEL
LIN {X 0,Y 354.891,Z 387.279,A -85,B 0,C 180,E1 -13345.828,E2 -13345.828} C_VEL
LIN {X 0,Y 354.845,Z 387.284,A -85,B 0,C 180,E1 -13349.679,E2 -13349.679} C_VEL
LIN {X 0,Y 354.821,Z 387.287,A -85,B 0,C 180,E1 -13353.683,E2 -13353.683} C_VEL
LIN {X 0,Y 354.793,Z 387.289,A -85,B 0,C 180,E1 -13356.46,E2 -13356.46} C_VEL
LIN {X 0,Y 354.816,Z 387.288,A -85,B 0,C 180,E1 -13359.425,E2 -13359.425} C_VEL
LIN {X 0,Y 354.782,Z 387.291,A -85,B 0,C 180,E1 -13362.869,E2 -13362.869} C_VEL
LIN {X 0,Y 354.769,Z 387.291,A -85,B 0,C 180,E1 -13366.107,E2 -13366.107} C_VEL
LIN {X 0,Y 354.782,Z 387.291,A -85,B 0,C 180,E1 -13369.181,E2 -13369.181} C_VEL
LIN {X 0,Y 354.803,Z 387.288,A -85,B 0,C 180,E1 -13372.404,E2 -13372.404} C_VEL
LIN {X 0,Y 354.808,Z 387.29,A -85,B 0,C 180,E1 -13374.942,E2 -13374.942} C_VEL
LIN {X 0,Y 354.811,Z 387.289,A -85,B 0,C 180,E1 -13378.401,E2 -13378.401} C_VEL
LIN {X 0,Y 354.869,Z 387.345,A -85,B 0,C 180,E1 -13380.121,E2 -13380.121} C_VEL
LIN {X 0,Y 357.202,Z 398.429,A -85,B 0,C 180,E1 -13383.096,E2 -13383.096} C_VEL
LIN {X 0,Y 358.552,Z 406.089,A -85,B 0,C 180,E1 -13385.077,E2 -13385.077} C_VEL
LIN {X 0,Y 358.316,Z 410.161,A -85,B 0,C 180,E1 -13386.042,E2 -13386.042} C_VEL
LIN {X 0,Y 363.097,Z 434.693,A -85,B 0,C 180,E1 -13387.238,E2 -13387.238} C_VEL
LIN {X 0,Y 365.301,Z 452.271,A -85,B 0,C 180,E1 -13387.946,E2 -13387.946} C_VEL
LIN {X 0,Y 362.82,Z 527.638,A -85,B 0,C 180,E1 -13389.892,E2 -13389.892} C_VEL
LIN {X 0,Y 361.923,Z 540.582,A -85,B 0,C 180,E1 -13390.431,E2 -13390.431} C_VEL
LIN {X 0,Y 360.957,Z 552.125,A -85,B 0,C 180,E1 -13391.115,E2 -13391.115} C_VEL
LIN {X 0,Y 359.742,Z 564.421,A -85,B 0,C 180,E1 -13392.081,E2 -13392.081} C_VEL
LIN {X 0,Y 358.523,Z 575.521,A -85,B 0,C 180,E1 -13393.195,E2 -13393.195} C_VEL
LIN {X 0,Y 357.308,Z 586.094,A -85,B 0,C 180,E1 -13394.536,E2 -13394.536} C_VEL
LIN {X 0,Y 356.274,Z 595.503,A -85,B 0,C 180,E1 -13396.018,E2 -13396.018} C_VEL
LIN {X 0,Y 355.317,Z 602.913,A -85,B 0,C 180,E1 -13397.435,E2 -13397.435} C_VEL
LIN {X 0,Y 354.47,Z 610.206,A -85,B 0,C 180,E1 -13399.145,E2 -13399.145} C_VEL
LIN {X 0,Y 353.873,Z 616.03,A -85,B 0,C 180,E1 -13400.86,E2 -13400.86} C_VEL
LIN {X 0,Y 353.51,Z 620.595,A -85,B 0,C 180,E1 -13402.577,E2 -13402.577} C_VEL
LIN {X 0,Y 353.259,Z 625.329,A -85,B 0,C 180,E1 -13404.865,E2 -13404.865} C_VEL
LIN {X 0,Y 353.222,Z 627.825,A -85,B 0,C 180,E1 -13406.579,E2 -13406.579} C_VEL
LIN {X 0,Y 353.173,Z 628.956,A -85,B 0,C 180,E1 -13407.721,E2 -13407.721} C_VEL
LIN {X 0,Y 353.217,Z 629.657,A -85,B 0,C 180,E1 -13408.861,E2 -13408.861} C_VEL
LIN {X 0,Y 353.261,Z 629.963,A -85,B 0,C 180,E1 -13410.001,E2 -13410.001} C_VEL
LIN {X 0,Y 353.203,Z 629.873,A -85,B 0,C 180,E1 -13411.142,E2 -13411.142} C_VEL
LIN {X 0,Y 353.171,Z 629.359,A -85,B 0,C 180,E1 -13412.282,E2 -13412.282} C_VEL
LIN {X 0,Y 353.219,Z 628.423,A -85,B 0,C 180,E1 -13413.424,E2 -13413.424} C_VEL
LIN {X 0,Y 353.264,Z 627.087,A -85,B 0,C 180,E1 -13414.566,E2 -13414.566} C_VEL
LIN {X 0,Y 353.297,Z 624.923,A -85,B 0,C 180,E1 -13415.938,E2 -13415.938} C_VEL
LIN {X 0,Y 353.624,Z 620.414,A -85,B 0,C 180,E1 -13417.998,E2 -13417.998} C_VEL
LIN {X 0,Y 354.063,Z 615.43,A -85,B 0,C 180,E1 -13419.715,E2 -13419.715} C_VEL
LIN {X 0,Y 354.711,Z 609.168,A -85,B 0,C 180,E1 -13421.429,E2 -13421.429} C_VEL
LIN {X 0,Y 355.746,Z 601.381,A -85,B 0,C 180,E1 -13423.133,E2 -13423.133} C_VEL
LIN {X 0,Y 356.732,Z 593.438,A -85,B 0,C 180,E1 -13424.549,E2 -13424.549} C_VEL
LIN {X 0,Y 357.778,Z 583.773,A -85,B 0,C 180,E1 -13425.964,E2 -13425.964} C_VEL
LIN {X 0,Y 359.007,Z 573.073,A -85,B 0,C 180,E1 -13427.224,E2 -13427.224} C_VEL
LIN {X 0,Y 360.157,Z 562.754,A -85,B 0,C 180,E1 -13428.194,E2 -13428.194} C_VEL
LIN {X 0,Y 361.255,Z 550.477,A -85,B 0,C 180,E1 -13429.093,E2 -13429.093} C_VEL
LIN {X 0,Y 362.257,Z 536.941,A -85,B 0,C 180,E1 -13429.811,E2 -13429.811} C_VEL
LIN {X 0,Y 363.018,Z 524.278,A -85,B 0,C 180,E1 -13430.248,E2 -13430.248} C_VEL
LIN {X 0,Y 364.491,Z 451.988,A -85,B 0,C 180,E1 -13431.802,E2 -13431.802} C_VEL
LIN {X 0,Y 361.156,Z 430.832,A -85,B 0,C 180,E1 -13432.534,E2 -13432.534} C_VEL
LIN {X 0,Y 358.409,Z 416.959,A -85,B 0,C 180,E1 -13433.091,E2 -13433.091} C_VEL
LIN {X 0,Y 359.258,Z 409.658,A -85,B 0,C 180,E1 -13434.874,E2 -13434.874} C_VEL
LIN {X 0,Y 358.632,Z 404.736,A -85,B 0,C 180,E1 -13436.183,E2 -13436.183} C_VEL
LIN {X 0,Y 356.455,Z 394.011,A -85,B 0,C 180,E1 -13439.209,E2 -13439.209} C_VEL
LIN {X 0,Y 354.82,Z 387.293,A -85,B 0,C 180,E1 -13441.272,E2 -13441.272} C_VEL
LIN {X 0,Y 354.817,Z 387.29,A -85,B 0,C 180,E1 -13445.06,E2 -13445.06} C_VEL
LIN {X 0,Y 354.811,Z 387.292,A -85,B 0,C 180,E1 -13447.884,E2 -13447.884} C_VEL
LIN {X 0,Y 354.793,Z 387.297,A -85,B 0,C 180,E1 -13451.172,E2 -13451.172} C_VEL
LIN {X 0,Y 354.769,Z 387.295,A -85,B 0,C 180,E1 -13454.507,E2 -13454.507} C_VEL
LIN {X 0,Y 354.8,Z 387.288,A -85,B 0,C 180,E1 -13457.663,E2 -13457.663} C_VEL
LIN {X 0,Y 354.821,Z 387.284,A -85,B 0,C 180,E1 -13460.667,E2 -13460.667} C_VEL
LIN {X 0,Y 354.827,Z 387.285,A -85,B 0,C 180,E1 -13464.301,E2 -13464.301} C_VEL
LIN {X 0,Y 354.793,Z 387.289,A -85,B 0,C 180,E1 -13467.667,E2 -13467.667} C_VEL
LIN {X 0,Y 354.852,Z 387.281,A -85,B 0,C 180,E1 -13471.619,E2 -13471.619} C_VEL
LIN {X 0,Y 354.905,Z 387.27,A -85,B 0,C 180,E1 -13474.173,E2 -13474.173} C_VEL
LIN {X 0,Y 354.842,Z 387.277,A -85,B 0,C 180,E1 -13477.894,E2 -13477.894} C_VEL
LIN {X 0,Y 354.929,Z 387.265,A -85,B 0,C 180,E1 -13481.892,E2 -13481.892} C_VEL
LIN {X 0,Y 354.949,Z 387.263,A -85,B 0,C 180,E1 -13485.982,E2 -13485.982} C_VEL
LIN {X 0,Y 354.984,Z 387.258,A -85,B 0,C 180,E1 -13489.736,E2 -13489.736} C_VEL
LIN {X 0,Y 355.121,Z 387.251,A -85,B 0,C 180,E1 -13492.037,E2 -13492.037} C_VEL
LIN {X 0,Y 355.099,Z 387.25,A -85,B 0,C 180,E1 -13494.321,E2 -13494.321} C_VEL
LIN {X 0,Y 355.25,Z 387.227,A -85,B 0,C 180,E1 -13497.733,E2 -13497.733} C_VEL
LIN {X 0,Y 355.381,Z 387.214,A -85,B 0,C 180,E1 -13500,E2 -13500} C_VEL
LIN {X 0,Y 355.25,Z 387.235,A -85,B 0,C 180,E1 -13502.268,E2 -13502.268} C_VEL
LIN {X 0,Y 355.145,Z 387.242,A -85,B 0,C 180,E1 -13506.819,E2 -13506.819} C_VEL
LIN {X 0,Y 355.022,Z 387.261,A -85,B 0,C 180,E1 -13509.112,E2 -13509.112} C_VEL
LIN {X 0,Y 354.928,Z 387.274,A -85,B 0,C 180,E1 -13512.581,E2 -13512.581} C_VEL
LIN {X 0,Y 354.896,Z 387.278,A -85,B 0,C 180,E1 -13516.096,E2 -13516.096} C_VEL
LIN {X 0,Y 354.913,Z 387.278,A -85,B 0,C 180,E1 -13518.472,E2 -13518.472} C_VEL
LIN {X 0,Y 354.841,Z 387.286,A -85,B 0,C 180,E1 -13522.106,E2 -13522.106} C_VEL
LIN {X 0,Y 354.89,Z 387.281,A -85,B 0,C 180,E1 -13524.73,E2 -13524.73} C_VEL
LIN {X 0,Y 357.184,Z 397.879,A -85,B 0,C 180,E1 -13528.179,E2 -13528.179} C_VEL
LIN {X 0,Y 357.677,Z 400.396,A -85,B 0,C 180,E1 -13528.938,E2 -13528.938} C_VEL
LIN {X 0,Y 361.724,Z 411.259,A -85,B 0,C 180,E1 -13529.511,E2 -13529.511} C_VEL
LIN {X 0,Y 365.007,Z 426.925,A -85,B 0,C 180,E1 -13530.121,E2 -13530.121} C_VEL
LIN {X 0,Y 363.102,Z 507.731,A -85,B 0,C 180,E1 -13531.863,E2 -13531.863} C_VEL
LIN {X 0,Y 362.461,Z 521.189,A -85,B 0,C 180,E1 -13532.385,E2 -13532.385} C_VEL
LIN {X 0,Y 361.667,Z 532.984,A -85,B 0,C 180,E1 -13533.051,E2 -13533.051} C_VEL
LIN {X 0,Y 360.643,Z 545.051,A -85,B 0,C 180,E1 -13533.972,E2 -13533.972} C_VEL
LIN {X 0,Y 359.515,Z 556.162,A -85,B 0,C 180,E1 -13535.064,E2 -13535.064} C_VEL
LIN {X 0,Y 358.442,Z 565.719,A -85,B 0,C 180,E1 -13536.231,E2 -13536.231} C_VEL
LIN {X 0,Y 357.31,Z 574.72,A -85,B 0,C 180,E1 -13537.571,E2 -13537.571} C_VEL
LIN {X 0,Y 356.266,Z 583.249,A -85,B 0,C 180,E1 -13539.143,E2 -13539.143} C_VEL
LIN {X 0,Y 355.367,Z 590.282,A -85,B 0,C 180,E1 -13540.741,E2 -13540.741} C_VEL
LIN {X 0,Y 354.628,Z 596.076,A -85,B 0,C 180,E1 -13542.362,E2 -13542.362} C_VEL
LIN {X 0,Y 353.948,Z 601.676,A -85,B 0,C 180,E1 -13544.37,E2 -13544.37} C_VEL
LIN {X 0,Y 353.628,Z 604.93,A -85,B 0,C 180,E1 -13545.924,E2 -13545.924} C_VEL
LIN {X 0,Y 353.299,Z 607.318,A -85,B 0,C 180,E1 -13547.44,E2 -13547.44} C_VEL
LIN {X 0,Y 353.116,Z 609.104,A -85,B 0,C 180,E1 -13549.14,E2 -13549.14} C_VEL
LIN {X 0,Y 352.979,Z 610.005,A -85,B 0,C 180,E1 -13550.943,E2 -13550.943} C_VEL
LIN {X 0,Y 352.958,Z 609.882,A -85,B 0,C 180,E1 -13552.795,E2 -13552.795} C_VEL
LIN {X 0,Y 353.054,Z 608.602,A -85,B 0,C 180,E1 -13554.739,E2 -13554.739} C_VEL
LIN {X 0,Y 353.307,Z 606.154,A -85,B 0,C 180,E1 -13556.665,E2 -13556.665} C_VEL
LIN {X 0,Y 353.717,Z 601.781,A -85,B 0,C 180,E1 -13558.895,E2 -13558.895} C_VEL
LIN {X 0,Y 354.152,Z 596.426,A -85,B 0,C 180,E1 -13560.829,E2 -13560.829} C_VEL
LIN {X 0,Y 354.814,Z 590.195,A -85,B 0,C 180,E1 -13562.578,E2 -13562.578} C_VEL
LIN {X 0,Y 355.526,Z 582.914,A -85,B 0,C 180,E1 -13564.22,E2 -13564.22} C_VEL
LIN {X 0,Y 356.492,Z 573.906,A -85,B 0,C 180,E1 -13565.852,E2 -13565.852} C_VEL
LIN {X 0,Y 357.445,Z 564.793,A -85,B 0,C 180,E1 -13567.187,E2 -13567.187} C_VEL
LIN {X 0,Y 358.405,Z 554.399,A -85,B 0,C 180,E1 -13568.427,E2 -13568.427} C_VEL
LIN {X 0,Y 359.378,Z 543.146,A -85,B 0,C 180,E1 -13569.498,E2 -13569.498} C_VEL
LIN {X 0,Y 360.179,Z 531.367,A -85,B 0,C 180,E1 -13570.364,E2 -13570.364} C_VEL
LIN {X 0,Y 360.939,Z 518.177,A -85,B 0,C 180,E1 -13571.074,E2 -13571.074} C_VEL
LIN {X 0,Y 361.453,Z 504.974,A -85,B 0,C 180,E1 -13571.543,E2 -13571.543} C_VEL
LIN {X 0,Y 362.998,Z 425.436,A -85,B 0,C 180,E1 -13573.216,E2 -13573.216} C_VEL
LIN {X 0,Y 358.665,Z 403.861,A -85,B 0,C 180,E1 -13573.94,E2 -13573.94} C_VEL
LIN {X 0,Y 357.163,Z 399.178,A -85,B 0,C 180,E1 -13574.155,E2 -13574.155} C_VEL
LIN {X 0,Y 355.107,Z 388.058,A -85,B 0,C 180,E1 -13577.424,E2 -13577.424} C_VEL
LIN {X 0,Y 354.948,Z 387.27,A -85,B 0,C 180,E1 -13577.709,E2 -13577.709} C_VEL
LIN {X 0,Y 355.003,Z 387.263,A -85,B 0,C 180,E1 -13580.886,E2 -13580.886} C_VEL
LIN {X 0,Y 355.081,Z 387.256,A -85,B 0,C 180,E1 -13584.319,E2 -13584.319} C_VEL
LIN {X 0,Y 355.248,Z 387.231,A -85,B 0,C 180,E1 -13587.731,E2 -13587.731} C_VEL
LIN {X 0,Y 355.4,Z 387.214,A -85,B 0,C 180,E1 -13589.999,E2 -13589.999} C_VEL
LIN {X 0,Y 355.249,Z 387.236,A -85,B 0,C 180,E1 -13592.266,E2 -13592.266} C_VEL
LIN {X 0,Y 355.141,Z 387.245,A -85,B 0,C 180,E1 -13596.818,E2 -13596.818} C_VEL
LIN {X 0,Y 354.993,Z 387.262,A -85,B 0,C 180,E1 -13599.417,E2 -13599.417} C_VEL
LIN {X 0,Y 354.923,Z 387.273,A -85,B 0,C 180,E1 -13602.579,E2 -13602.579} C_VEL
LIN {X 0,Y 354.926,Z 387.273,A -85,B 0,C 180,E1 -13604.353,E2 -13604.353} C_VEL
LIN {X 0,Y 354.242,Z 387.357,A -85,B 0,C 180,E1 -13605.3,E2 -13605.3} C_VEL
LIN {X 0,Y 351.386,Z 387.712,A -85,B 0,C 180,E1 -13606.842,E2 -13606.842} C_VEL
LIN {X 0,Y 348.965,Z 388.018,A -85,B 0,C 180,E1 -13608.089,E2 -13608.089} C_VEL
LIN {X 0,Y 347.911,Z 388.144,A -85,B 0,C 180,E1 -13609.054,E2 -13609.054} C_VEL
LIN {X 0,Y 347.817,Z 388.156,A -85,B 0,C 180,E1 -13609.381,E2 -13609.381} C_VEL
LIN {X 0,Y 347.766,Z 388.163,A -85,B 0,C 180,E1 -13612.578,E2 -13612.578} C_VEL
LIN {X 0,Y 347.809,Z 388.157,A -85,B 0,C 180,E1 -13615.107,E2 -13615.107} C_VEL
LIN {X 0,Y 347.811,Z 388.162,A -85,B 0,C 180,E1 -13617.692,E2 -13617.692} C_VEL
LIN {X 0,Y 347.769,Z 388.163,A -85,B 0,C 180,E1 -13620.344,E2 -13620.344} C_VEL
LIN {X 0,Y 347.744,Z 388.168,A -85,B 0,C 180,E1 -13624.042,E2 -13624.042} C_VEL
LIN {X 0,Y 347.762,Z 388.166,A -85,B 0,C 180,E1 -13627.318,E2 -13627.318} C_VEL
LIN {X 0,Y 347.75,Z 388.165,A -85,B 0,C 180,E1 -13630.292,E2 -13630.292} C_VEL
LIN {X 0,Y 347.832,Z 388.365,A -85,B 0,C 180,E1 -13633.889,E2 -13633.889} C_VEL
LIN {X 0,Y 349.737,Z 397.883,A -85,B 0,C 180,E1 -13636.099,E2 -13636.099} C_VEL
LIN {X 0,Y 351.703,Z 405.943,A -85,B 0,C 180,E1 -13636.408,E2 -13636.408} C_VEL
LIN {X 0,Y 355.168,Z 426.079,A -85,B 0,C 180,E1 -13637.092,E2 -13637.092} C_VEL
LIN {X 0,Y 353.106,Z 507.36,A -85,B 0,C 180,E1 -13639.055,E2 -13639.055} C_VEL
LIN {X 0,Y 352.671,Z 519.382,A -85,B 0,C 180,E1 -13639.541,E2 -13639.541} C_VEL
LIN {X 0,Y 351.956,Z 532.149,A -85,B 0,C 180,E1 -13640.283,E2 -13640.283} C_VEL
LIN {X 0,Y 351.152,Z 544.363,A -85,B 0,C 180,E1 -13641.231,E2 -13641.231} C_VEL
LIN {X 0,Y 350.353,Z 554.944,A -85,B 0,C 180,E1 -13642.278,E2 -13642.278} C_VEL
LIN {X 0,Y 349.444,Z 565.33,A -85,B 0,C 180,E1 -13643.557,E2 -13643.557} C_VEL
LIN {X 0,Y 348.658,Z 574.489,A -85,B 0,C 180,E1 -13644.936,E2 -13644.936} C_VEL
LIN {X 0,Y 347.846,Z 583.437,A -85,B 0,C 180,E1 -13646.594,E2 -13646.594} C_VEL
LIN {X 0,Y 347.258,Z 590.629,A -85,B 0,C 180,E1 -13648.25,E2 -13648.25} C_VEL
LIN {X 0,Y 346.695,Z 597.276,A -85,B 0,C 180,E1 -13650.169,E2 -13650.169} C_VEL
LIN {X 0,Y 346.367,Z 602.535,A -85,B 0,C 180,E1 -13652.18,E2 -13652.18} C_VEL
LIN {X 0,Y 346.204,Z 605.142,A -85,B 0,C 180,E1 -13653.474,E2 -13653.474} C_VEL
LIN {X 0,Y 346.016,Z 607.13,A -85,B 0,C 180,E1 -13654.752,E2 -13654.752} C_VEL
LIN {X 0,Y 345.926,Z 608.661,A -85,B 0,C 180,E1 -13656.093,E2 -13656.093} C_VEL
LIN {X 0,Y 345.865,Z 609.536,A -85,B 0,C 180,E1 -13657.289,E2 -13657.289} C_VEL
LIN {X 0,Y 345.918,Z 610.004,A -85,B 0,C 180,E1 -13659.155,E2 -13659.155} C_VEL
LIN {X 0,Y 346.064,Z 609.378,A -85,B 0,C 180,E1 -13661.038,E2 -13661.038} C_VEL
LIN {X 0,Y 346.266,Z 608.115,A -85,B 0,C 180,E1 -13662.535,E2 -13662.535} C_VEL
LIN {X 0,Y 346.661,Z 604.932,A -85,B 0,C 180,E1 -13664.719,E2 -13664.719} C_VEL
LIN {X 0,Y 347.099,Z 601.45,A -85,B 0,C 180,E1 -13666.375,E2 -13666.375} C_VEL
LIN {X 0,Y 347.91,Z 595.948,A -85,B 0,C 180,E1 -13668.346,E2 -13668.346} C_VEL
LIN {X 0,Y 348.864,Z 589.24,A -85,B 0,C 180,E1 -13670.199,E2 -13670.199} C_VEL
LIN {X 0,Y 349.999,Z 581.388,A -85,B 0,C 180,E1 -13671.92,E2 -13671.92} C_VEL
LIN {X 0,Y 351.169,Z 573.115,A -85,B 0,C 180,E1 -13673.392,E2 -13673.392} C_VEL
LIN {X 0,Y 352.419,Z 563.644,A -85,B 0,C 180,E1 -13674.766,E2 -13674.766} C_VEL
LIN {X 0,Y 353.902,Z 551.584,A -85,B 0,C 180,E1 -13676.157,E2 -13676.157} C_VEL
LIN {X 0,Y 355.067,Z 540.476,A -85,B 0,C 180,E1 -13677.164,E2 -13677.164} C_VEL
LIN {X 0,Y 356.195,Z 527.175,A -85,B 0,C 180,E1 -13678.092,E2 -13678.092} C_VEL
LIN {X 0,Y 357.095,Z 514.321,A -85,B 0,C 180,E1 -13678.731,E2 -13678.731} C_VEL
LIN {X 0,Y 357.72,Z 500.327,A -85,B 0,C 180,E1 -13679.184,E2 -13679.184} C_VEL
LIN {X 0,Y 360.346,Z 427.542,A -85,B 0,C 180,E1 -13681.055,E2 -13681.055} C_VEL
LIN {X 0,Y 357.272,Z 413.282,A -85,B 0,C 180,E1 -13681.786,E2 -13681.786} C_VEL
LIN {X 0,Y 352.602,Z 402.442,A -85,B 0,C 180,E1 -13682.613,E2 -13682.613} C_VEL
LIN {X 0,Y 350.974,Z 398.933,A -85,B 0,C 180,E1 -13682.927,E2 -13682.927} C_VEL
LIN {X 0,Y 348.051,Z 388.136,A -85,B 0,C 180,E1 -13685.867,E2 -13685.867} C_VEL
LIN {X 0,Y 348.083,Z 388.125,A -85,B 0,C 180,E1 -13688.388,E2 -13688.388} C_VEL
LIN {X 0,Y 347.883,Z 388.151,A -85,B 0,C 180,E1 -13692.84,E2 -13692.84} C_VEL
LIN {X 0,Y 347.831,Z 388.159,A -85,B 0,C 180,E1 -13696.432,E2 -13696.432} C_VEL
LIN {X 0,Y 347.853,Z 388.155,A -85,B 0,C 180,E1 -13698.86,E2 -13698.86} C_VEL
LIN {X 0,Y 347.83,Z 388.158,A -85,B 0,C 180,E1 -13701.657,E2 -13701.657} C_VEL
LIN {X 0,Y 347.812,Z 388.159,A -85,B 0,C 180,E1 -13705.108,E2 -13705.108} C_VEL
LIN {X 0,Y 347.803,Z 388.162,A -85,B 0,C 180,E1 -13707.695,E2 -13707.695} C_VEL
LIN {X 0,Y 347.761,Z 388.167,A -85,B 0,C 180,E1 -13710.347,E2 -13710.347} C_VEL
LIN {X 0,Y 347.739,Z 388.17,A -85,B 0,C 180,E1 -13714.045,E2 -13714.045} C_VEL
LIN {X 0,Y 347.757,Z 388.166,A -85,B 0,C 180,E1 -13717.321,E2 -13717.321} C_VEL
LIN {X 0,Y 347.725,Z 388.17,A -85,B 0,C 180,E1 -13720.298,E2 -13720.298} C_VEL
LIN {X 0,Y 347.718,Z 388.174,A -85,B 0,C 180,E1 -13723.409,E2 -13723.409} C_VEL
